								eRFID[iw1].lrWeightMeasuredCV := eWeightPackageState[1].lrWeightMeasuredCV := VIS.lrWeight1Measured;
								eRFID[iw1].lrWeightCV := eWeightPackageState[1].lrWeightCV := VIS.lrWeight1Mass:=P05_Weight.fbWeight1.lrMeasuredWeight+lrWeight1MeasurmentCorrection-lrCupWeight-lrFormWeight-lrFormWeight1RFID;	
								
								(***DIAGNOSTYKA WAGI***)
									IF eRFID[iw1].lrMinWeightCV = 0 THEN eRFID[iw1].lrMinWeightCV := ABS(eRFID[iw1].lrWeightCV); END_IF
									IF eRFID[iw1].lrMinWeightCV > ABS(eRFID[iw1].lrWeightCV)  THEN
											eRFID[iw1].lrMinWeightCV:= ABS(eRFID[iw1].lrWeightCV);
									END_IF
									IF ABS(eRFID[iw1].lrWeightCV) > eRFID[iw1].lrMaxWeightCV THEN
											eRFID[iw1].lrMaxWeightCV:= ABS(eRFID[iw1].lrWeightCV);
									END_IF
									eRFID[iw1].lrWeightDif := eRFID[iw1].lrMaxWeightCV - eRFID[iw1].lrMinWeightCV;
								(***KONIEC DIAGNOSTYKI WAGI**)
								
							
								eRFID[iw1].lrWeightSV := eWeightPackageState[1].lrWeightSV := lrWeightMassSV;
								eRFID[iw1].bWeighed := eWeightPackageState[1].bWeighed := TRUE;
								//Sprawdzanie czy doza spełnia kryteria dopuszczalenej konfekcji
								
								(*Generowaie danych do wykresów*)
								IF eRFID[iw1].nDispencerNr = 1 THEN
									VIS.lrDispencer1WeightMeasured := eRFID[iw1].lrWeightCV;	//Do wykresów HMI
									VIS.lrDispencer1DoseVolumeCV :=	eRFID[iw1].lrDoseVolumeCV;	//Do wykresów HMI
									VIS.bDispencer1WeightMeasured := TRUE; //Do wyświetlenia na ekranie głównym
								ELSE									  
									VIS.lrDispencer1WeightMeasured := VIS.lrDispencer1DoseVolumeCV := 0.0;	//Do wykresów HMI
									VIS.bDispencer1WeightMeasured := FALSE; //Do wyświetlenia na ekranie głównym
								END_IF
							
								(*Koniec generowania danych do wykresów*)
								IF 	((LREAL_TO_DINT(eRFID[iw1].lrWeightCV)-LREAL_TO_DINT(eRFID[iw1].lrWeightSV))<=(lrWeightUpperTolerance)) AND 
									((LREAL_TO_DINT(eRFID[iw1].lrWeightSV)-LREAL_TO_DINT(eRFID[iw1].lrWeightCV))<=lrWeightLowerTolerance) 
									THEN
									eRFID[iw1].bWeightOK := eWeightPackageState[1].bWeightOK := TRUE;
								END_IF	
								(*Dodatkowa informacja o wadze*)
								IF 	((LREAL_TO_DINT(eRFID[iw1].lrWeightCV)-LREAL_TO_DINT(eRFID[iw1].lrWeightSV))>lrWeightUpperTolerance) THEN
									eRFID[iw1].bWeightTooHigh := eWeightPackageState[1].bWeightTooHigh := TRUE;
								END_IF
								IF ((LREAL_TO_DINT(eRFID[iw1].lrWeightSV)-LREAL_TO_DINT(eRFID[iw1].lrWeightCV))>lrWeightLowerTolerance) THEN
									eRFID[iw1].bWeightTooLow:= eWeightPackageState[1].bWeightTooLow := TRUE;
								END_IF				
								VIS.bWeight1DoWeighting:=FALSE;
								
							END_IF																		
						ELSIF NOT bWeight1Enable THEN
							eRFID[iw1].bWeightOK 			:= eWeightPackageState[1].bWeightOK 			:=	TRUE;
							eRFID[iw1].bWeightTooHigh 		:= eWeightPackageState[1].bWeightTooHigh 		:=	FALSE;
							eRFID[iw1].bWeightTooLow		:= eWeightPackageState[1].bWeightTooLow 		:=	FALSE;
							eRFID[iw1].lrWeightMeasuredCV 	:= eWeightPackageState[1].lrWeightMeasuredCV 	:=	0;
							eRFID[iw1].lrWeightCV 			:= eWeightPackageState[1].lrWeightCV 			:=	VIS.lrWeight1Mass:=lrWeightMassSV;	
							eRFID[iw1].lrWeightSV 			:= eWeightPackageState[1].lrWeightSV 			:=	lrWeightMassSV;
							eRFID[iw1].bWeighed 			:= eWeightPackageState[1].bWeighed  			:=	FALSE;
						END_IF
						//KONIEC WARUNKI STACJI								
				ELSIF tonWeightPackageState1BnCardNumber0.Q THEN	// Jeżeli nie wykryje RFID
					VIS.bWeight1DoWeighting 			:= FALSE;
					eWeightPackageState[1].bFormPresent	:= TRUE;					
					eWeightPackageState[1].bWeightOK	:= FALSE;
					eWeightPackageState[1].bWeighed		:= TRUE;
				ELSIF tonWeightPackageState1BnNoCardNumber.Q THEN 	// Jeżeli nie ma RFID w tablicy
					itonWeightPackageState1BnNoCardNumber	:= itonWeightPackageState1BnNoCardNumber	+	1;
					VIS.bWeight1DoWeighting 			:= FALSE;
					eWeightPackageState[1].bWeightOK 	:= FALSE;
					eWeightPackageState[1].bWeighed 	:= TRUE;
				ELSE
					;
				END_IF
				
			END_FOR	
		END_IF

// Waga 2
tonWeightPackageState2BnCardNumber0			(IN:=eWeightPackageState[2].nCardNumber = 0 AND VIS.bWeight2DoWeighting OR NOT bWeight1Enable, PT:=T#5S);
tonWeightPackageState2BnNoCardNumber		(IN:=eWeightPackageState[2].nCardNumber > 0 AND VIS.bWeight2DoWeighting OR NOT bWeight1Enable, PT:=T#10S);
IF VIS.bWeight2DoWeighting THEN
			FOR iw2 := 1 TO 100 DO
				 IF eWeightPackageState[2].nCardNumber = eRFID[iw2].nCardNumber AND eWeightPackageState[2].nCardNumber > 0 THEN	
						nw2:=iw2; (*Do testów*) eRFID[nw2].bFormPresent; eRFID[nw2].bWeighed; eRFID[nw2].lrWeightMeasuredCV;
				 		//WARUNKI STACJI
						IF bWeight1Enable AND  NOT eRFID[iw2].bWeighed AND eRFID[iw2].lrWeightMeasuredCV=0 
						THEN
							//VIS.bWeight2Run:=TRUE;
							IF P05_Weight.fbWeight2.bCycleDone THEN	
								//(*Włączona waga z przeważania*) // Czyli w recepturach waga formatki wybrana na 0
								IF lrFormWeight = 0 THEN
											FOR jw2 := 1 TO 100 DO
												IF eWeightPackageState[2].nCardNumber = VIS.AnRFIDCardNumberShow[jw2] THEN	
													lrFormWeight2RFID := VIS.AnRFIDWeightShow[jw2];
													bFormWeight2Found := TRUE;
												END_IF
											END_FOR
											IF NOT bFormWeight2Found THEN
												lrFormWeight2RFID := 0;
											END_IF
											bFormWeight2Found := FALSE;
								ELSE
									lrFormWeight2RFID := 0;
								END_IF
								(**KONIEC POBIERANIE WARTOŚCI Z PRZEWAŻANIA*)
						
								eRFID[iw2].lrWeightMeasuredCV := eWeightPackageState[2].lrWeightMeasuredCV := VIS.lrWeight2Measured;
								eRFID[iw2].lrWeightCV := eWeightPackageState[2].lrWeightCV := VIS.lrWeight2Mass:=P05_Weight.fbWeight2.lrMeasuredWeight+lrWeight1MeasurmentCorrection-lrCupWeight-lrFormWeight-lrFormWeight2RFID;	
								
								(***DIAGNOSTYKA WAGI***)
									IF eRFID[iw2].lrMinWeightCV = 0 THEN eRFID[iw2].lrMinWeightCV := ABS(eRFID[iw2].lrWeightCV); END_IF
									IF eRFID[iw2].lrMinWeightCV > ABS(eRFID[iw2].lrWeightCV)  THEN
											eRFID[iw2].lrMinWeightCV:= ABS(eRFID[iw2].lrWeightCV);
									END_IF
									IF ABS(eRFID[iw2].lrWeightCV) > eRFID[iw2].lrMaxWeightCV THEN
											eRFID[iw2].lrMaxWeightCV:= ABS(eRFID[iw2].lrWeightCV);
									END_IF
									eRFID[iw2].lrWeightDif := eRFID[iw2].lrMaxWeightCV - eRFID[iw2].lrMinWeightCV;
								(***KONIEC DIAGNOSTYKI WAGI**)
								
							
								eRFID[iw2].lrWeightSV := eWeightPackageState[2].lrWeightSV := lrWeightMassSV;
								eRFID[iw2].bWeighed := eWeightPackageState[2].bWeighed:= TRUE;
								//Sprawdzanie czy doza spełnia kryteria dopuszczalenej konfekcji
								
								(*Generowaie danych do wykresów*)
								(*IF eRFID[iw2].nDispencerNr = 1 THEN
									VIS.lrDispencer1WeightMeasured := eRFID[iw2].lrWeightCV;	//Do wykresów HMI
									VIS.lrDispencer1DoseVolumeCV :=	eRFID[iw2].lrDoseVolumeCV;	//Do wykresów HMI
									VIS.bDispencer1WeightMeasured := TRUE; //Do wyświetlenia na ekranie głównym
								ELSE									  
									VIS.lrDispencer1WeightMeasured := VIS.lrDispencer1DoseVolumeCV := 0.0;	//Do wykresów HMI
									VIS.bDispencer1WeightMeasured := FALSE; //Do wyświetlenia na ekranie głównym
								END_IF*)
								IF eRFID[iw2].nDispencerNr = 2 THEN
									VIS.lrDispencer2WeightMeasured := eRFID[iw2].lrWeightCV;	//Do wykresów HMI
									VIS.lrDispencer2DoseVolumeCV :=	eRFID[iw2].lrDoseVolumeCV;	//Do wykresów HMI
									VIS.bDispencer2WeightMeasured := TRUE; //Do wyświetlenia na ekranie głównym
									IF bDosingTwoPhases THEN
										VIS.lrDispencer2DoseVolumeCV :=	eRFID[iw2].lrDoseVolumeCVSecondPhase; //Do wykresów HMI
									END_IF
								ELSE									
									VIS.lrDispencer2WeightMeasured := VIS.lrDispencer2DoseVolumeCV := 0.0;	//Do wykresów HMI
									VIS.bDispencer2WeightMeasured := FALSE; //Do wyświetlenia na ekranie głównym
								END_IF
								(*IF eRFID[iw2].nDispencerNr = 3 THEN
									VIS.lrDispencer3WeightMeasured := eRFID[iw2].lrWeightCV;	//Do wykresów HMI
									VIS.lrDispencer3DoseVolumeCV :=	eRFID[iw2].lrDoseVolumeCV;	//Do wykresów HMI
									VIS.bDispencer3WeightMeasured := TRUE; //Do wyświetlenia na ekranie głównym
								ELSE									  
									VIS.lrDispencer3WeightMeasured := VIS.lrDispencer3DoseVolumeCV := 0.0;	//Do wykresów HMI
									VIS.bDispencer3WeightMeasured := FALSE; //Do wyświetlenia na ekranie głównym
								END_IF
								
								IF eRFID[iw2].nDispencerNr = 4 THEN
									VIS.lrDispencer4WeightMeasured := eRFID[iw2].lrWeightCV;	//Do wykresów HMI
									VIS.lrDispencer4DoseVolumeCV :=	eRFID[iw2].lrDoseVolumeCV;	//Do wykresów HMI
									VIS.bDispencer4WeightMeasured := TRUE; //Do wyświetlenia na ekranie głównym
								ELSE									  
									VIS.lrDispencer4WeightMeasured := VIS.lrDispencer4DoseVolumeCV := 0.0;	//Do wykresów HMI
									VIS.bDispencer4WeightMeasured := FALSE; //Do wyświetlenia na ekranie głównym
								END_IF*)
								(*Koniec generowania danych do wykresów*)
								IF 	((LREAL_TO_DINT(eRFID[iw2].lrWeightCV)-LREAL_TO_DINT(eRFID[iw2].lrWeightSV))<=(lrWeightUpperTolerance)) AND 
									((LREAL_TO_DINT(eRFID[iw2].lrWeightSV)-LREAL_TO_DINT(eRFID[iw2].lrWeightCV))<=lrWeightLowerTolerance) 
									THEN
									eRFID[iw2].bWeightOK := eWeightPackageState[2].bWeightOK := TRUE;
								END_IF	
								(*Dodatkowa informacja o wadze*)
								IF 	((LREAL_TO_DINT(eRFID[iw2].lrWeightCV)-LREAL_TO_DINT(eRFID[iw2].lrWeightSV))>lrWeightUpperTolerance) THEN
									eRFID[iw2].bWeightTooHigh := eWeightPackageState[2].bWeightTooHigh := TRUE;
								END_IF
								IF ((LREAL_TO_DINT(eRFID[iw2].lrWeightSV)-LREAL_TO_DINT(eRFID[iw2].lrWeightCV))>lrWeightLowerTolerance) THEN
									eRFID[iw2].bWeightTooLow:= eWeightPackageState[2].bWeightTooLow := TRUE;
								END_IF	
								
								VIS.bWeight2DoWeighting:=FALSE;
								
							END_IF																		
						ELSIF NOT bWeight1Enable THEN
							eRFID[iw2].bWeightOK := eWeightPackageState[2].bWeightOK := TRUE;
							eRFID[iw2].bWeightTooHigh := eWeightPackageState[2].bWeightTooHigh := FALSE;
							eRFID[iw2].bWeightTooLow:= eWeightPackageState[2].bWeightTooLow := FALSE;
							eRFID[iw2].lrWeightMeasuredCV := eWeightPackageState[2].lrWeightMeasuredCV := 0;
							eRFID[iw2].lrWeightCV := eWeightPackageState[2].lrWeightCV :=VIS.lrWeight2Mass:=lrWeightMassSV;	
							eRFID[iw2].lrWeightSV := eWeightPackageState[2].lrWeightSV :=lrWeightMassSV;
							eRFID[iw2].bWeighed := eWeightPackageState[2].bWeighed  := FALSE;
						END_IF
						//KONIEC WARUNKI STACJI								
				ELSIF tonWeightPackageState2BnCardNumber0.Q THEN	// Jeżeli nie wykryje RFID
					VIS.bWeight2DoWeighting 					:= FALSE;
					eWeightPackageState[2].bFormPresent	:= TRUE;	//Dp		
					eWeightPackageState[2].bWeightOK	:= FALSE;
					eWeightPackageState[2].bWeighed		:= TRUE;
				ELSIF tonWeightPackageState2BnNoCardNumber.Q THEN 	// Jeżeli nie ma RFID w tablicy
					itonWeightPackageState2BnNoCardNumber	:= itonWeightPackageState2BnNoCardNumber	+	1;					
					VIS.bWeight2DoWeighting 					:= FALSE;
					eWeightPackageState[2].bWeightOK 	:= FALSE;
					eWeightPackageState[2].bWeighed 	:= TRUE;
				ELSE
					;
				END_IF
				
			END_FOR	
		END_IF

// Waga 3
tonWeightPackageState3BnCardNumber0			(IN:=eWeightPackageState[3].nCardNumber = 0 AND VIS.bWeight3DoWeighting OR NOT bWeight1Enable, PT:=T#5S);
tonWeightPackageState3BnNoCardNumber		(IN:=eWeightPackageState[3].nCardNumber > 0 AND VIS.bWeight3DoWeighting OR NOT bWeight1Enable, PT:=T#10S);
IF VIS.bWeight3DoWeighting THEN
			FOR iw3 := 1 TO 100 DO
				 IF eWeightPackageState[3].nCardNumber = eRFID[iw3].nCardNumber AND eWeightPackageState[3].nCardNumber > 0 THEN	
						nw3:=iw3; (*Do testów*) eRFID[nw3].bFormPresent; eRFID[nw3].bWeighed; eRFID[nw3].lrWeightMeasuredCV;
				 		//WARUNKI STACJI
						IF bWeight1Enable AND NOT eRFID[iw3].bWeighed AND eRFID[iw3].lrWeightMeasuredCV=0 
						THEN
						//	VIS.bWeight3Run:=TRUE;
							IF P05_Weight.fbWeight3.bCycleDone THEN	
								//(*Włączona waga z przeważania*) // Czyli w recepturach waga formatki wybrana na 0
								IF lrFormWeight = 0 THEN
											FOR jw3 := 1 TO 100 DO
												IF eWeightPackageState[3].nCardNumber = VIS.AnRFIDCardNumberShow[jw3] THEN	
													lrFormWeight3RFID := VIS.AnRFIDWeightShow[jw3];
													bFormWeight3Found := TRUE;
												END_IF
											END_FOR
											IF NOT bFormWeight3Found THEN
												lrFormWeight3RFID := 0;
											END_IF
											bFormWeight3Found := FALSE;
								ELSE
									lrFormWeight3RFID := 0;
								END_IF
								(**KONIEC POBIERANIE WARTOŚCI Z PRZEWAŻANIA*)
						
								eRFID[iw3].lrWeightMeasuredCV := eWeightPackageState[3].lrWeightMeasuredCV := VIS.lrWeight3Measured;
								eRFID[iw3].lrWeightCV := eWeightPackageState[3].lrWeightCV := VIS.lrWeight3Mass:=P05_Weight.fbWeight3.lrMeasuredWeight+lrWeight1MeasurmentCorrection-lrCupWeight-lrFormWeight-lrFormWeight3RFID;	
								
								(***DIAGNOSTYKA WAGI***)
									IF eRFID[iw3].lrMinWeightCV = 0 THEN eRFID[iw3].lrMinWeightCV := ABS(eRFID[iw3].lrWeightCV); END_IF
									IF eRFID[iw3].lrMinWeightCV > ABS(eRFID[iw3].lrWeightCV)  THEN
											eRFID[iw3].lrMinWeightCV:= ABS(eRFID[iw3].lrWeightCV);
									END_IF
									IF ABS(eRFID[iw3].lrWeightCV) > eRFID[iw3].lrMaxWeightCV THEN
											eRFID[iw3].lrMaxWeightCV:= ABS(eRFID[iw3].lrWeightCV);
									END_IF
									eRFID[iw3].lrWeightDif := eRFID[iw3].lrMaxWeightCV - eRFID[iw3].lrMinWeightCV;
								(***KONIEC DIAGNOSTYKI WAGI**)
								
							
								eRFID[iw3].lrWeightSV := eWeightPackageState[3].lrWeightSV := lrWeightMassSV;
								eRFID[iw3].bWeighed := eWeightPackageState[3].bWeighed := TRUE;
								//Sprawdzanie czy doza spełnia kryteria dopuszczalenej konfekcji
								
								(*Generowaie danych do wykresów*)
								(*IF eRFID[iw3].nDispencerNr = 1 THEN
									VIS.lrDispencer1WeightMeasured := eRFID[iw3].lrWeightCV;	//Do wykresów HMI
									VIS.lrDispencer1DoseVolumeCV :=	eRFID[iw3].lrDoseVolumeCV;	//Do wykresów HMI
									VIS.bDispencer1WeightMeasured := TRUE; //Do wyświetlenia na ekranie głównym
								ELSE									  
									VIS.lrDispencer1WeightMeasured := VIS.lrDispencer1DoseVolumeCV := 0.0;	//Do wykresów HMI
									VIS.bDispencer1WeightMeasured := FALSE; //Do wyświetlenia na ekranie głównym
								END_IF
								IF eRFID[iw3].nDispencerNr = 2 THEN
									VIS.lrDispencer2WeightMeasured := eRFID[iw3].lrWeightCV;	//Do wykresów HMI
									VIS.lrDispencer2DoseVolumeCV :=	eRFID[iw3].lrDoseVolumeCV;	//Do wykresów HMI
									VIS.bDispencer2WeightMeasured := TRUE; //Do wyświetlenia na ekranie głównym
									IF bDosingTwoPhases THEN
										VIS.lrDispencer2DoseVolumeCV :=	eRFID[iw3].lrDoseVolumeCVSecondPhase; //Do wykresów HMI
									END_IF
								ELSE									
									VIS.lrDispencer2WeightMeasured := VIS.lrDispencer2DoseVolumeCV := 0.0;	//Do wykresów HMI
									VIS.bDispencer2WeightMeasured := FALSE; //Do wyświetlenia na ekranie głównym
								END_IF*)
								IF eRFID[iw3].nDispencerNr = 3 THEN
									VIS.lrDispencer3WeightMeasured := eRFID[iw3].lrWeightCV;	//Do wykresów HMI
									VIS.lrDispencer3DoseVolumeCV :=	eRFID[iw3].lrDoseVolumeCV;	//Do wykresów HMI
									VIS.bDispencer3WeightMeasured := TRUE; //Do wyświetlenia na ekranie głównym
								ELSE									  
									VIS.lrDispencer3WeightMeasured := VIS.lrDispencer3DoseVolumeCV := 0.0;	//Do wykresów HMI
									VIS.bDispencer3WeightMeasured := FALSE; //Do wyświetlenia na ekranie głównym
								END_IF
								
								(*IF eRFID[iw3].nDispencerNr = 4 THEN
									VIS.lrDispencer4WeightMeasured := eRFID[iw3].lrWeightCV;	//Do wykresów HMI
									VIS.lrDispencer4DoseVolumeCV :=	eRFID[iw3].lrDoseVolumeCV;	//Do wykresów HMI
									VIS.bDispencer4WeightMeasured := TRUE; //Do wyświetlenia na ekranie głównym
								ELSE									  
									VIS.lrDispencer4WeightMeasured := VIS.lrDispencer4DoseVolumeCV := 0.0;	//Do wykresów HMI
									VIS.bDispencer4WeightMeasured := FALSE; //Do wyświetlenia na ekranie głównym
								END_IF	*)						
								(*Koniec generowania danych do wykresów*)
								IF 	((LREAL_TO_DINT(eRFID[iw3].lrWeightCV)-LREAL_TO_DINT(eRFID[iw3].lrWeightSV))<=(lrWeightUpperTolerance)) AND 
									((LREAL_TO_DINT(eRFID[iw3].lrWeightSV)-LREAL_TO_DINT(eRFID[iw3].lrWeightCV))<=lrWeightLowerTolerance) 
									THEN
									eRFID[iw3].bWeightOK := eWeightPackageState[3].bWeightOK := TRUE;
								END_IF	
								(*Dodatkowa informacja o wadze*)
								
								IF 	((LREAL_TO_DINT(eRFID[iw3].lrWeightCV)-LREAL_TO_DINT(eRFID[iw3].lrWeightSV))>lrWeightUpperTolerance) THEN
									eRFID[iw3].bWeightTooHigh := eWeightPackageState[3].bWeightTooHigh := TRUE;
								END_IF
								IF ((LREAL_TO_DINT(eRFID[iw3].lrWeightSV)-LREAL_TO_DINT(eRFID[iw3].lrWeightCV))>lrWeightLowerTolerance) THEN
									eRFID[iw3].bWeightTooLow:= eWeightPackageState[3].bWeightTooLow := TRUE;
								END_IF	
								
								VIS.bWeight3DoWeighting:=FALSE;
								
							END_IF																		
						ELSIF NOT bWeight1Enable THEN
							eRFID[iw3].bWeightOK := eWeightPackageState[3].bWeightOK := TRUE;
							eRFID[iw3].bWeightTooHigh := eWeightPackageState[3].bWeightTooHigh := FALSE;
							eRFID[iw3].bWeightTooLow:= eWeightPackageState[3].bWeightTooLow := FALSE;
							eRFID[iw3].lrWeightMeasuredCV := eWeightPackageState[3].lrWeightMeasuredCV := 0;
							eRFID[iw3].lrWeightCV := eWeightPackageState[3].lrWeightCV :=VIS.lrWeight3Mass:=lrWeightMassSV;	
							eRFID[iw3].lrWeightSV := eWeightPackageState[3].lrWeightSV :=lrWeightMassSV;
							eRFID[iw3].bWeighed := eWeightPackageState[3].bWeighed  := FALSE;
						END_IF
						//KONIEC WARUNKI STACJI								
				ELSIF tonWeightPackageState3BnCardNumber0.Q THEN	// Jeżeli nie wykryje RFID
					VIS.bWeight3DoWeighting 					:= FALSE;
					eWeightPackageState[3].bFormPresent	:= TRUE;	//Dp		
					eWeightPackageState[3].bWeightOK 	:= FALSE;
					eWeightPackageState[3].bWeighed 	:= TRUE;
				ELSIF tonWeightPackageState3BnNoCardNumber.Q THEN 	// Jeżeli nie ma RFID w tablicy
					itonWeightPackageState3BnNoCardNumber	:= itonWeightPackageState3BnNoCardNumber	+	1;						
					VIS.bWeight3DoWeighting 					:= FALSE;
					eWeightPackageState[3].bWeightOK 	:= FALSE;
					eWeightPackageState[3].bWeighed 	:= TRUE;
				ELSE
					;
				END_IF
				
			END_FOR	
		END_IF

// Waga 4
tonWeightPackageState4BnCardNumber0			(IN:=eWeightPackageState[4].nCardNumber = 0 AND VIS.bWeight4DoWeighting OR NOT bWeight1Enable, PT:=T#5S);
tonWeightPackageState4BnNoCardNumber		(IN:=eWeightPackageState[4].nCardNumber > 0 AND VIS.bWeight4DoWeighting OR NOT bWeight1Enable, PT:=T#10S);
IF VIS.bWeight4DoWeighting THEN
			FOR iw4 := 1 TO 100 DO
				 IF eWeightPackageState[4].nCardNumber = eRFID[iw4].nCardNumber AND eWeightPackageState[4].nCardNumber > 0 THEN	
						nw4:=iw4; (*Do testów*) eRFID[nw4].bFormPresent; eRFID[nw4].bWeighed; eRFID[nw4].lrWeightMeasuredCV;
				 		//WARUNKI STACJI
						IF bWeight1Enable AND NOT eRFID[iw4].bWeighed AND eRFID[iw4].lrWeightMeasuredCV=0 
						THEN
							//VIS.bWeight4Run:=TRUE;
							IF P05_Weight.fbWeight4.bCycleDone THEN	
								//(*Włączona waga z przeważania*) // Czyli w recepturach waga formatki wybrana na 0
								IF lrFormWeight = 0 THEN
											FOR jw4 := 1 TO 100 DO
												IF eWeightPackageState[4].nCardNumber = VIS.AnRFIDCardNumberShow[jw4] THEN	
													lrFormWeight4RFID := VIS.AnRFIDWeightShow[jw4];
													bFormWeight4Found := TRUE;
												END_IF
											END_FOR
											IF NOT bFormWeight4Found THEN
												lrFormWeight4RFID := 0;
											END_IF
											bFormWeight4Found := FALSE;
								ELSE
									lrFormWeight4RFID := 0;
								END_IF
								(**KONIEC POBIERANIE WARTOŚCI Z PRZEWAŻANIA*)
						
								eRFID[iw4].lrWeightMeasuredCV := eWeightPackageState[4].lrWeightMeasuredCV := VIS.lrWeight4Measured;
								eRFID[iw4].lrWeightCV := eWeightPackageState[4].lrWeightCV := VIS.lrWeight4Mass:=P05_Weight.fbWeight4.lrMeasuredWeight+lrWeight1MeasurmentCorrection-lrCupWeight-lrFormWeight-lrFormWeight4RFID;	
								
								(***DIAGNOSTYKA WAGI***)
									IF eRFID[iw4].lrMinWeightCV = 0 THEN eRFID[iw4].lrMinWeightCV := ABS(eRFID[iw4].lrWeightCV); END_IF
									IF eRFID[iw4].lrMinWeightCV > ABS(eRFID[iw4].lrWeightCV)  THEN
											eRFID[iw4].lrMinWeightCV:= ABS(eRFID[iw4].lrWeightCV);
									END_IF
									IF ABS(eRFID[iw4].lrWeightCV) > eRFID[iw4].lrMaxWeightCV THEN
											eRFID[iw4].lrMaxWeightCV:= ABS(eRFID[iw4].lrWeightCV);
									END_IF
									eRFID[iw4].lrWeightDif := eRFID[iw4].lrMaxWeightCV - eRFID[iw4].lrMinWeightCV;
								(***KONIEC DIAGNOSTYKI WAGI**)
								
							
								eRFID[iw4].lrWeightSV := eWeightPackageState[4].lrWeightSV := lrWeightMassSV;
								eRFID[iw4].bWeighed := eWeightPackageState[4].bWeighed := TRUE;
								//Sprawdzanie czy doza spełnia kryteria dopuszczalenej konfekcji
								
								(*Generowaie danych do wykresów*)
								(*IF eRFID[iw4].nDispencerNr = 1 THEN
									VIS.lrDispencer1WeightMeasured := eRFID[iw4].lrWeightCV;	//Do wykresów HMI
									VIS.lrDispencer1DoseVolumeCV :=	eRFID[iw4].lrDoseVolumeCV;	//Do wykresów HMI
									VIS.bDispencer1WeightMeasured := TRUE; //Do wyświetlenia na ekranie głównym
								ELSE									  
									VIS.lrDispencer1WeightMeasured := VIS.lrDispencer1DoseVolumeCV := 0.0;	//Do wykresów HMI
									VIS.bDispencer1WeightMeasured := FALSE; //Do wyświetlenia na ekranie głównym
								END_IF
								IF eRFID[iw4].nDispencerNr = 2 THEN
									VIS.lrDispencer2WeightMeasured := eRFID[iw4].lrWeightCV;	//Do wykresów HMI
									VIS.lrDispencer2DoseVolumeCV :=	eRFID[iw4].lrDoseVolumeCV;	//Do wykresów HMI
									VIS.bDispencer2WeightMeasured := TRUE; //Do wyświetlenia na ekranie głównym
									IF bDosingTwoPhases THEN
										VIS.lrDispencer2DoseVolumeCV :=	eRFID[iw4].lrDoseVolumeCVSecondPhase; //Do wykresów HMI
									END_IF
								ELSE									
									VIS.lrDispencer2WeightMeasured := VIS.lrDispencer2DoseVolumeCV := 0.0;	//Do wykresów HMI
									VIS.bDispencer2WeightMeasured := FALSE; //Do wyświetlenia na ekranie głównym
								END_IF
								IF eRFID[iw4].nDispencerNr = 3 THEN
									VIS.lrDispencer3WeightMeasured := eRFID[iw4].lrWeightCV;	//Do wykresów HMI
									VIS.lrDispencer3DoseVolumeCV :=	eRFID[iw4].lrDoseVolumeCV;	//Do wykresów HMI
									VIS.bDispencer3WeightMeasured := TRUE; //Do wyświetlenia na ekranie głównym
								ELSE									  
									VIS.lrDispencer3WeightMeasured := VIS.lrDispencer3DoseVolumeCV := 0.0;	//Do wykresów HMI
									VIS.bDispencer3WeightMeasured := FALSE; //Do wyświetlenia na ekranie głównym
								END_IF*)
								
								IF eRFID[iw4].nDispencerNr = 4 THEN
									VIS.lrDispencer4WeightMeasured := eRFID[iw4].lrWeightCV;	//Do wykresów HMI
									VIS.lrDispencer4DoseVolumeCV :=	eRFID[iw4].lrDoseVolumeCV;	//Do wykresów HMI
									VIS.bDispencer4WeightMeasured := TRUE; //Do wyświetlenia na ekranie głównym
								ELSE									  
									VIS.lrDispencer4WeightMeasured := VIS.lrDispencer4DoseVolumeCV := 0.0;	//Do wykresów HMI
									VIS.bDispencer4WeightMeasured := FALSE; //Do wyświetlenia na ekranie głównym
								END_IF
								
								(*Koniec generowania danych do wykresów*)
								IF 	((LREAL_TO_DINT(eRFID[iw4].lrWeightCV)-LREAL_TO_DINT(eRFID[iw4].lrWeightSV))<=(lrWeightUpperTolerance)) AND 
									((LREAL_TO_DINT(eRFID[iw4].lrWeightSV)-LREAL_TO_DINT(eRFID[iw4].lrWeightCV))<=lrWeightLowerTolerance) 
									THEN
									eRFID[iw4].bWeightOK := eWeightPackageState[4].bWeightOK := TRUE;
								END_IF	
								(*Dodatkowa informacja o wadze*)
								IF 	((LREAL_TO_DINT(eRFID[iw4].lrWeightCV)-LREAL_TO_DINT(eRFID[iw4].lrWeightSV))>lrWeightUpperTolerance) THEN
									eRFID[iw4].bWeightTooHigh := eWeightPackageState[4].bWeightTooHigh := TRUE;
								END_IF
								IF ((LREAL_TO_DINT(eRFID[iw4].lrWeightSV)-LREAL_TO_DINT(eRFID[iw4].lrWeightCV))>lrWeightLowerTolerance) THEN
									eRFID[iw4].bWeightTooLow:= eWeightPackageState[4].bWeightTooLow := TRUE;
								END_IF

							VIS.bWeight4DoWeighting:=FALSE;
	
							END_IF																		
						ELSIF NOT bWeight1Enable THEN
							eRFID[iw4].bWeightOK := eWeightPackageState[4].bWeightOK := TRUE;
							eRFID[iw4].bWeightTooHigh := eWeightPackageState[4].bWeightTooHigh := FALSE;
							eRFID[iw4].bWeightTooLow:= eWeightPackageState[4].bWeightTooLow := FALSE;
							eRFID[iw4].lrWeightMeasuredCV := eWeightPackageState[4].lrWeightMeasuredCV := 0;
							eRFID[iw4].lrWeightCV := eWeightPackageState[4].lrWeightCV :=VIS.lrWeight4Mass:=lrWeightMassSV;	
							eRFID[iw4].lrWeightSV := eWeightPackageState[4].lrWeightSV :=lrWeightMassSV;
							eRFID[iw4].bWeighed := eWeightPackageState[4].bWeighed  := FALSE;
						END_IF
						//KONIEC WARUNKI STACJI								
				ELSIF tonWeightPackageState4BnCardNumber0.Q THEN	// Jeżeli nie wykryje RFID
					VIS.bWeight4DoWeighting 					:= FALSE;
					eWeightPackageState[4].bFormPresent	:= TRUE;	//Dp		
					eWeightPackageState[4].bWeightOK 	:= FALSE;
					eWeightPackageState[4].bWeighed 	:= TRUE;
				ELSIF tonWeightPackageState4BnNoCardNumber.Q THEN 	// Jeżeli nie ma RFID w tablicy
					itonWeightPackageState4BnNoCardNumber	:= itonWeightPackageState4BnNoCardNumber	+	1;							
					VIS.bWeight4DoWeighting 					:= FALSE;
					eWeightPackageState[4].bWeightOK 	:= FALSE;
					eWeightPackageState[4].bWeighed 	:= TRUE;
				ELSE
					;
				END_IF
				
			END_FOR	
		END_IF										
(********************KONIEC WAZENIA**************************)
(************************************************************)

(********************Ważenie przy dwufazie**************************)
(*******************************************************************)






// Waga 5 - 1 waga na drugiej fazie
tonWeightPackageState5BnCardNumber0			(IN:=eWeightPackage2PhasePackageState[1].nCardNumber = 0 AND VIS.bWeight5DoWeighting OR NOT bWeight1Enable, PT:=T#3S);
tonWeightPackageState5BnNoCardNumber		(IN:=eWeightPackage2PhasePackageState[1].nCardNumber > 0 AND VIS.bWeight5DoWeighting OR NOT bWeight1Enable, PT:=T#10S);
IF VIS.bWeight5DoWeighting THEN
			FOR iw5 := 1 TO 100 DO
				 IF eWeightPackage2PhasePackageState[1].nCardNumber = eRFID[iw5].nCardNumber AND eWeightPackage2PhasePackageState[1].nCardNumber > 0 THEN	
						nw5:=iw5; (*Do testów*) eRFID[nw5].bFormPresent; eRFID[nw5].bWeighed; eRFID[nw5].lrWeightMeasuredCV;
				 		//WARUNKI STACJI
						IF bWeight1Enable AND NOT eRFID[iw5].bWeighed AND eRFID[iw5].lrWeightMeasuredCV=0 
						THEN
							//VIS.bWeight4Run:=TRUE;
							IF P05_Weight.fbWeight5.bCycleDone THEN	
								//(*Włączona waga z przeważania*) // Czyli w recepturach waga formatki wybrana na 0
								IF lrFormWeight = 0 THEN
											FOR jw5 := 1 TO 100 DO
												IF eWeightPackage2PhasePackageState[1].nCardNumber = VIS.AnRFIDCardNumberShow[jw5] THEN	
													lrFormWeight5RFID := VIS.AnRFIDWeightShow[jw5];
													bFormWeight5Found := TRUE;
												END_IF
											END_FOR
											IF NOT bFormWeight5Found THEN
												lrFormWeight5RFID := 0;
											END_IF
											bFormWeight5Found := FALSE;
								ELSE
									lrFormWeight5RFID := 0;
								END_IF
								(**KONIEC POBIERANIE WARTOŚCI Z PRZEWAŻANIA*)
						
								eRFID[iw5].lrWeightMeasuredCV := eWeightPackage2PhasePackageState[1].lrWeightMeasuredCV := VIS.lrWeight5Measured;
								eRFID[iw5].lrWeightCV := eWeightPackage2PhasePackageState[1].lrWeightCV := VIS.lrWeight5Mass:=P05_Weight.fbWeight5.lrMeasuredWeight+lrWeight1MeasurmentCorrection-lrCupWeight-lrFormWeight-lrFormWeight5RFID;	
								
								(***DIAGNOSTYKA WAGI***)
									IF eRFID[iw5].lrMinWeightCV = 0 THEN eRFID[iw5].lrMinWeightCV := ABS(eRFID[iw5].lrWeightCV); END_IF
									IF eRFID[iw5].lrMinWeightCV > ABS(eRFID[iw5].lrWeightCV)  THEN
											eRFID[iw5].lrMinWeightCV:= ABS(eRFID[iw5].lrWeightCV);
									END_IF
									IF ABS(eRFID[iw5].lrWeightCV) > eRFID[iw5].lrMaxWeightCV THEN
											eRFID[iw5].lrMaxWeightCV:= ABS(eRFID[iw5].lrWeightCV);
									END_IF
									eRFID[iw5].lrWeightDif := eRFID[iw5].lrMaxWeightCV - eRFID[iw5].lrMinWeightCV;
								(***KONIEC DIAGNOSTYKI WAGI**)
								
							
								eRFID[iw5].lrWeightSV := eWeightPackage2PhasePackageState[1].lrWeightSV := lrWeightMassSV;
								eRFID[iw5].bWeighed := eWeightPackage2PhasePackageState[1].bWeighed := TRUE;
								//Sprawdzanie czy doza spełnia kryteria dopuszczalenej konfekcji
								
								(*Generowaie danych do wykresów*)
								VIS.lrDispencer1WeightMeasured 	:= eRFID[iw5].lrWeightCV;	//Do wykresów HMI
								//VIS.lrDispencer1DoseVolumeCV 	:=	eRFID[iw5].lrDoseVolumeCV;	//Do wykresów HMI
								
								IF eRFID[iw5].nDispencerNr = 1 THEN
									VIS.lrDispencer1DoseVolumeCV :=	eRFID[iw5].lrDoseVolumeCV;	
								ELSIF eRFID[iw5].nDispencerNr = 2 THEN
									VIS.lrDispencer2DoseVolumeCV :=	eRFID[iw5].lrDoseVolumeCV;
								ELSIF eRFID[iw5].nDispencerNr = 3 THEN
									VIS.lrDispencer3DoseVolumeCV :=	eRFID[iw5].lrDoseVolumeCVSecondPhase;
								ELSIF eRFID[iw5].nDispencerNr = 4 THEN
									VIS.lrDispencer4DoseVolumeCV :=	eRFID[iw5].lrDoseVolumeCVSecondPhase;	
								ELSE									  
									VIS.lrDispencer4DoseVolumeCV := 0.0;
								END_IF	
			
								(*IF eRFID[iw5].nDispencerNr = 1 THEN
									VIS.lrDispencer1WeightMeasured := eRFID[iw5].lrWeightCV;	//Do wykresów HMI
									VIS.lrDispencer1DoseVolumeCV :=	eRFID[iw5].lrDoseVolumeCV;	//Do wykresów HMI
									VIS.bDispencer1WeightMeasured := TRUE; //Do wyświetlenia na ekranie głównym
								ELSE									  
									VIS.lrDispencer1WeightMeasured := VIS.lrDispencer1DoseVolumeCV := 0.0;	//Do wykresów HMI
									VIS.bDispencer1WeightMeasured := FALSE; //Do wyświetlenia na ekranie głównym
								END_IF
								IF eRFID[iw5].nDispencerNr = 2 THEN
									VIS.lrDispencer2WeightMeasured := eRFID[iw5].lrWeightCV;	//Do wykresów HMI
									VIS.lrDispencer2DoseVolumeCV :=	eRFID[iw5].lrDoseVolumeCV;	//Do wykresów HMI
									VIS.bDispencer2WeightMeasured := TRUE; //Do wyświetlenia na ekranie głównym
									IF bDosingTwoPhases THEN
										VIS.lrDispencer2DoseVolumeCV :=	eRFID[iw5].lrDoseVolumeCVSecondPhase; //Do wykresów HMI
									END_IF
								ELSE									
									VIS.lrDispencer2WeightMeasured := VIS.lrDispencer2DoseVolumeCV := 0.0;	//Do wykresów HMI
									VIS.bDispencer2WeightMeasured := FALSE; //Do wyświetlenia na ekranie głównym
								END_IF
								IF eRFID[iw5].nDispencerNr = 3 THEN
									VIS.lrDispencer3WeightMeasured := eRFID[iw5].lrWeightCV;	//Do wykresów HMI
									VIS.lrDispencer3DoseVolumeCV :=	eRFID[iw5].lrDoseVolumeCV;	//Do wykresów HMI
									VIS.bDispencer3WeightMeasured := TRUE; //Do wyświetlenia na ekranie głównym
								ELSE									  
									VIS.lrDispencer3WeightMeasured := VIS.lrDispencer3DoseVolumeCV := 0.0;	//Do wykresów HMI
									VIS.bDispencer3WeightMeasured := FALSE; //Do wyświetlenia na ekranie głównym
								END_IF
								
								IF eRFID[iw5].nDispencerNr = 4 THEN
									VIS.lrDispencer4WeightMeasured := eRFID[iw5].lrWeightCV;	//Do wykresów HMI
									VIS.lrDispencer4DoseVolumeCV :=	eRFID[iw5].lrDoseVolumeCV;	//Do wykresów HMI
									VIS.bDispencer4WeightMeasured := TRUE; //Do wyświetlenia na ekranie głównym
								ELSE									  
									VIS.lrDispencer4WeightMeasured := VIS.lrDispencer4DoseVolumeCV := 0.0;	//Do wykresów HMI
									VIS.bDispencer4WeightMeasured := FALSE; //Do wyświetlenia na ekranie głównym
								END_IF*)
								
								
								
								(*Koniec generowania danych do wykresów*)
								IF 	((LREAL_TO_DINT(eRFID[iw5].lrWeightCV)-LREAL_TO_DINT(eRFID[iw5].lrWeightSV))<=(lrWeightUpperTolerance)) AND 
									((LREAL_TO_DINT(eRFID[iw5].lrWeightSV)-LREAL_TO_DINT(eRFID[iw5].lrWeightCV))<=lrWeightLowerTolerance) 
									THEN
									eRFID[iw5].bWeightOK := eWeightPackage2PhasePackageState[1].bWeightOK := TRUE;
								END_IF	
								(*Dodatkowa informacja o wadze*)
								IF 	((LREAL_TO_DINT(eRFID[iw5].lrWeightCV)-LREAL_TO_DINT(eRFID[iw5].lrWeightSV))>lrWeightUpperTolerance) THEN
									eRFID[iw5].bWeightTooHigh := eWeightPackage2PhasePackageState[1].bWeightTooHigh := TRUE;
								END_IF
								IF ((LREAL_TO_DINT(eRFID[iw5].lrWeightSV)-LREAL_TO_DINT(eRFID[iw5].lrWeightCV))>lrWeightLowerTolerance) THEN
									eRFID[iw5].bWeightTooLow:= eWeightPackage2PhasePackageState[1].bWeightTooLow := TRUE;
								END_IF

							VIS.bWeight5DoWeighting:=FALSE;
	
							END_IF																		
						ELSIF NOT bWeight1Enable THEN
							eRFID[iw5].bWeightOK := eWeightPackage2PhasePackageState[1].bWeightOK := TRUE;
							eRFID[iw5].bWeightTooHigh := eWeightPackage2PhasePackageState[1].bWeightTooHigh := FALSE;
							eRFID[iw5].bWeightTooLow:= eWeightPackage2PhasePackageState[1].bWeightTooLow := FALSE;
							eRFID[iw5].lrWeightMeasuredCV := eWeightPackage2PhasePackageState[1].lrWeightMeasuredCV := 0;
							eRFID[iw5].lrWeightCV := eWeightPackage2PhasePackageState[1].lrWeightCV :=VIS.lrWeight5Mass:=lrWeightMassSV;	
							eRFID[iw5].lrWeightSV := eWeightPackage2PhasePackageState[1].lrWeightSV :=lrWeightMassSV;
							eRFID[iw5].bWeighed := eWeightPackage2PhasePackageState[1].bWeighed  := FALSE;
						END_IF
						//KONIEC WARUNKI STACJI								
				ELSIF tonWeightPackageState5BnCardNumber0.Q THEN	// Jeżeli nie wykryje RFID
					VIS.bWeight5DoWeighting 					:= FALSE;
					eWeightPackage2PhasePackageState[1].bFormPresent	:= TRUE;	//Dp		
					eWeightPackage2PhasePackageState[1].bWeightOK 	:= FALSE;
					eWeightPackage2PhasePackageState[1].bWeighed 	:= TRUE;
				ELSIF tonWeightPackageState5BnNoCardNumber.Q THEN 	// Jeżeli nie ma RFID w tablicy
					VIS.bWeight5DoWeighting 					:= FALSE;
					eWeightPackage2PhasePackageState[1].bWeightOK 	:= FALSE;
					eWeightPackage2PhasePackageState[1].bWeighed 	:= TRUE;
				ELSE
					;
				END_IF
				
			END_FOR	
		END_IF	

// Waga 6 - 2 waga na drugiej fazie
tonWeightPackageState6BnCardNumber0			(IN:=eWeightPackage2PhasePackageState[2].nCardNumber = 0 AND VIS.bWeight6DoWeighting OR NOT bWeight1Enable, PT:=T#3S);
tonWeightPackageState6BnNoCardNumber		(IN:=eWeightPackage2PhasePackageState[2].nCardNumber > 0 AND VIS.bWeight6DoWeighting OR NOT bWeight1Enable, PT:=T#10S);
IF VIS.bWeight6DoWeighting THEN
			FOR iw6 := 1 TO 100 DO
				 IF eWeightPackage2PhasePackageState[2].nCardNumber = eRFID[iw6].nCardNumber AND eWeightPackage2PhasePackageState[2].nCardNumber > 0 THEN	
						nw6:=iw6; (*Do testów*) eRFID[nw6].bFormPresent; eRFID[nw6].bWeighed; eRFID[nw6].lrWeightMeasuredCV;
				 		//WARUNKI STACJI
						IF bWeight1Enable AND NOT eRFID[iw6].bWeighed AND eRFID[iw6].lrWeightMeasuredCV=0 
						THEN
							//VIS.bWeight4Run:=TRUE;
							IF P05_Weight.fbWeight6.bCycleDone THEN	
								//(*Włączona waga z przeważania*) // Czyli w recepturach waga formatki wybrana na 0
								IF lrFormWeight = 0 THEN
											FOR jw6 := 1 TO 100 DO
												IF eWeightPackage2PhasePackageState[2].nCardNumber = VIS.AnRFIDCardNumberShow[jw6] THEN	
													lrFormWeight6RFID := VIS.AnRFIDWeightShow[jw6];
													bFormWeight6Found := TRUE;
												END_IF
											END_FOR
											IF NOT bFormWeight6Found THEN
												lrFormWeight6RFID := 0;
											END_IF
											bFormWeight6Found := FALSE;
								ELSE
									lrFormWeight6RFID := 0;
								END_IF
								(**KONIEC POBIERANIE WARTOŚCI Z PRZEWAŻANIA*)
						
								eRFID[iw6].lrWeightMeasuredCV := eWeightPackage2PhasePackageState[2].lrWeightMeasuredCV := VIS.lrWeight6Measured;
								eRFID[iw6].lrWeightCV := eWeightPackage2PhasePackageState[2].lrWeightCV := VIS.lrWeight6Mass:=P05_Weight.fbWeight6.lrMeasuredWeight+lrWeight1MeasurmentCorrection-lrCupWeight-lrFormWeight-lrFormWeight6RFID;	
								
								(***DIAGNOSTYKA WAGI***)
									IF eRFID[iw6].lrMinWeightCV = 0 THEN eRFID[iw6].lrMinWeightCV := ABS(eRFID[iw6].lrWeightCV); END_IF
									IF eRFID[iw6].lrMinWeightCV > ABS(eRFID[iw6].lrWeightCV)  THEN
											eRFID[iw6].lrMinWeightCV:= ABS(eRFID[iw6].lrWeightCV);
									END_IF
									IF ABS(eRFID[iw6].lrWeightCV) > eRFID[iw6].lrMaxWeightCV THEN
											eRFID[iw6].lrMaxWeightCV:= ABS(eRFID[iw6].lrWeightCV);
									END_IF
									eRFID[iw6].lrWeightDif := eRFID[iw6].lrMaxWeightCV - eRFID[iw6].lrMinWeightCV;
								(***KONIEC DIAGNOSTYKI WAGI**)
								
							
								eRFID[iw6].lrWeightSV := eWeightPackage2PhasePackageState[2].lrWeightSV := lrWeightMassSV;
								eRFID[iw6].bWeighed := eWeightPackage2PhasePackageState[2].bWeighed := TRUE;
								//Sprawdzanie czy doza spełnia kryteria dopuszczalenej konfekcji
								
								(*Generowaie danych do wykresów*)
								
								VIS.lrDispencer2WeightMeasured 	:= eRFID[iw6].lrWeightCV;	//Do wykresów HMI
								//VIS.lrDispencer2DoseVolumeCV 	:= eRFID[iw6].lrDoseVolumeCV;	//Do wykresów HMI
								IF eRFID[iw6].nDispencerNr = 1 THEN
									VIS.lrDispencer1DoseVolumeCV :=	eRFID[iw6].lrDoseVolumeCV;	
								ELSIF eRFID[iw6].nDispencerNr = 2 THEN
									VIS.lrDispencer2DoseVolumeCV :=	eRFID[iw6].lrDoseVolumeCV;
								ELSIF eRFID[iw6].nDispencerNr = 3 THEN
									VIS.lrDispencer3DoseVolumeCV :=	eRFID[iw6].lrDoseVolumeCVSecondPhase;							
								ELSIF eRFID[iw6].nDispencerNr = 4 THEN
									VIS.lrDispencer4DoseVolumeCV :=	eRFID[iw6].lrDoseVolumeCVSecondPhase;	
								ELSE									  
									VIS.lrDispencer4DoseVolumeCV := 0.0;
								END_IF	
							
								(*IF eRFID[iw6].nDispencerNr = 1 THEN
									VIS.lrDispencer1WeightMeasured := eRFID[iw6].lrWeightCV;	//Do wykresów HMI
									VIS.lrDispencer1DoseVolumeCV :=	eRFID[iw6].lrDoseVolumeCV;	//Do wykresów HMI
									VIS.bDispencer1WeightMeasured := TRUE; //Do wyświetlenia na ekranie głównym
								ELSE									  
									VIS.lrDispencer1WeightMeasured := VIS.lrDispencer1DoseVolumeCV := 0.0;	//Do wykresów HMI
									VIS.bDispencer1WeightMeasured := FALSE; //Do wyświetlenia na ekranie głównym
								END_IF
								IF eRFID[iw6].nDispencerNr = 2 THEN
									VIS.lrDispencer2WeightMeasured := eRFID[iw6].lrWeightCV;	//Do wykresów HMI
									VIS.lrDispencer2DoseVolumeCV :=	eRFID[iw6].lrDoseVolumeCV;	//Do wykresów HMI
									VIS.bDispencer2WeightMeasured := TRUE; //Do wyświetlenia na ekranie głównym
									IF bDosingTwoPhases THEN
										VIS.lrDispencer2DoseVolumeCV :=	eRFID[iw6].lrDoseVolumeCVSecondPhase; //Do wykresów HMI
									END_IF
								ELSE									
									VIS.lrDispencer2WeightMeasured := VIS.lrDispencer2DoseVolumeCV := 0.0;	//Do wykresów HMI
									VIS.bDispencer2WeightMeasured := FALSE; //Do wyświetlenia na ekranie głównym
								END_IF
								IF eRFID[iw5].nDispencerNr = 3 THEN
									VIS.lrDispencer3WeightMeasured := eRFID[iw6].lrWeightCV;	//Do wykresów HMI
									VIS.lrDispencer3DoseVolumeCV :=	eRFID[iw6].lrDoseVolumeCV;	//Do wykresów HMI
									VIS.bDispencer3WeightMeasured := TRUE; //Do wyświetlenia na ekranie głównym
								ELSE									  
									VIS.lrDispencer3WeightMeasured := VIS.lrDispencer3DoseVolumeCV := 0.0;	//Do wykresów HMI
									VIS.bDispencer3WeightMeasured := FALSE; //Do wyświetlenia na ekranie głównym
								END_IF
								
								IF eRFID[iw6].nDispencerNr = 4 THEN
									VIS.lrDispencer4WeightMeasured := eRFID[iw6].lrWeightCV;	//Do wykresów HMI
									VIS.lrDispencer4DoseVolumeCV :=	eRFID[iw6].lrDoseVolumeCV;	//Do wykresów HMI
									VIS.bDispencer4WeightMeasured := TRUE; //Do wyświetlenia na ekranie głównym
								ELSE									  
									VIS.lrDispencer4WeightMeasured := VIS.lrDispencer4DoseVolumeCV := 0.0;	//Do wykresów HMI
									VIS.bDispencer4WeightMeasured := FALSE; //Do wyświetlenia na ekranie głównym
								END_IF*)
								
								(*Koniec generowania danych do wykresów*)
								IF 	((LREAL_TO_DINT(eRFID[iw6].lrWeightCV)-LREAL_TO_DINT(eRFID[iw6].lrWeightSV))<=(lrWeightUpperTolerance)) AND 
									((LREAL_TO_DINT(eRFID[iw6].lrWeightSV)-LREAL_TO_DINT(eRFID[iw6].lrWeightCV))<=lrWeightLowerTolerance) 
									THEN
									eRFID[iw6].bWeightOK := eWeightPackage2PhasePackageState[2].bWeightOK := TRUE;
								END_IF	
								(*Dodatkowa informacja o wadze*)
								IF 	((LREAL_TO_DINT(eRFID[iw6].lrWeightCV)-LREAL_TO_DINT(eRFID[iw6].lrWeightSV))>lrWeightUpperTolerance) THEN
									eRFID[iw6].bWeightTooHigh := eWeightPackage2PhasePackageState[2].bWeightTooHigh := TRUE;
								END_IF
								IF ((LREAL_TO_DINT(eRFID[iw6].lrWeightSV)-LREAL_TO_DINT(eRFID[iw6].lrWeightCV))>lrWeightLowerTolerance) THEN
									eRFID[iw6].bWeightTooLow:= eWeightPackage2PhasePackageState[2].bWeightTooLow := TRUE;
								END_IF

							VIS.bWeight6DoWeighting:=FALSE;
	
							END_IF																		
						ELSIF NOT bWeight1Enable THEN
							eRFID[iw6].bWeightOK := eWeightPackage2PhasePackageState[2].bWeightOK := TRUE;
							eRFID[iw6].bWeightTooHigh := eWeightPackage2PhasePackageState[2].bWeightTooHigh := FALSE;
							eRFID[iw6].bWeightTooLow:= eWeightPackage2PhasePackageState[2].bWeightTooLow := FALSE;
							eRFID[iw6].lrWeightMeasuredCV := eWeightPackage2PhasePackageState[2].lrWeightMeasuredCV := 0;
							eRFID[iw6].lrWeightCV := eWeightPackage2PhasePackageState[2].lrWeightCV :=VIS.lrWeight6Mass:=lrWeightMassSV;	
							eRFID[iw6].lrWeightSV := eWeightPackage2PhasePackageState[2].lrWeightSV :=lrWeightMassSV;
							eRFID[iw6].bWeighed := eWeightPackage2PhasePackageState[2].bWeighed  := FALSE;
						END_IF
						//KONIEC WARUNKI STACJI								
				ELSIF tonWeightPackageState6BnCardNumber0.Q THEN	// Jeżeli nie wykryje RFID
					VIS.bWeight6DoWeighting 					:= FALSE;
					eWeightPackage2PhasePackageState[2].bFormPresent	:= TRUE;	//Dp	
					eWeightPackage2PhasePackageState[2].bWeightOK 	:= FALSE;
					eWeightPackage2PhasePackageState[2].bWeighed 	:= TRUE;
				ELSIF tonWeightPackageState6BnNoCardNumber.Q THEN 	// Jeżeli nie ma RFID w tablicy
					VIS.bWeight6DoWeighting 					:= FALSE;
					eWeightPackage2PhasePackageState[2].bWeightOK 	:= FALSE;
					eWeightPackage2PhasePackageState[2].bWeighed 	:= TRUE;
				ELSE
					;
				END_IF
				
			END_FOR	
		END_IF
END_ACTION

ACTION aP05_WeightBlock:

IF bLidFeederEnable OR bWickFeederEnable THEN
	IF 
	eBeforeLidFeeder2PackageState[4].bFormPresent OR
	eBeforeLidFeeder2PackageState[3].bFormPresent OR
	eBeforeLidFeeder2PackageState[2].bFormPresent //OR
	//eBeforeLidFeeder2PackageState[1].bFormPresent	
	THEN
		bWeight1234ReleaseBlock := TRUE;
	ELSE
		bWeight1234ReleaseBlock := FALSE;
	END_IF

ELSE
	bWeight1234ReleaseBlock :=	FALSE;
END_IF



IF bDosingTwoPhases THEN
	IF ((*MAIN.IbLidSealerAfterSensor OR*) MAIN.IbLidSealerSecondFormSensor OR MAIN.IbLidFeederAfterSensor) AND (P00_PackML.fbPMLAuto.ePMLState = E_PMLState.ePMLState_EXECUTE)
	THEN
		bWeight56ReleaseBlock := TRUE;
	ELSE
		bWeight56ReleaseBlock := FALSE;
	END_IF

ELSE
	bWeight56ReleaseBlock :=	FALSE;
END_IF
END_ACTION

ACTION aP05_WeightGateBefore:
(*
Nazwa:			aP05_WeightGateBefore
Opis:			Szlabany przed wagą
Wersja:			v0.1
Data:			2024-04-09
Autor:			DP
Urzadzenia:		
Konfiguracja:	
Info:
*)
toWeightRealeseByLidFeeder (IN:= 	(	
										(
										NOT P05_Weight.fbIbWeight1FormBeforeSensor.bOUT AND
										NOT P05_Weight.fbIbWeight2FormBeforeSensor.bOUT AND
										NOT P05_Weight.fbIbWeight3FormBeforeSensor.bOUT AND
										NOT P05_Weight.fbIbWeight4FormBeforeSensor.bOUT AND 
										NOT P05_Weight.tonIbWeight1FormSensor.Q
										) OR
										NOT bLidFeederEnable
									), PT := T#50MS);




VIS.bGateBeforeWeight14Run;
VIS.bGateBeforeWeight56Run;
toniWeight14GateBeforeCASE	(IN:=	iWeightGateBeforeCASE = 60, PT:=T#0MS);
tonbGateBeforeWeight14Run	(IN:=	NOT eAfterDispencersPackageState[1].bFormPresent AND 
									NOT eAfterDispencersPackageState[2].bFormPresent AND 
									NOT eAfterDispencersPackageState[3].bFormPresent AND 
									NOT eAfterDispencersPackageState[4].bFormPresent 
									,PT:=T#100MS);
toniWeight14GateBeforeCASE2	(IN:=	iWeightGateBeforeCASE = 50 AND 
									eAfterDispencersPackageState[1].bFormPresent AND 
									eAfterDispencersPackageState[2].bFormPresent AND 
									eAfterDispencersPackageState[3].bFormPresent AND 
									eAfterDispencersPackageState[4].bFormPresent AND 
									VIS.bGateBeforeWeight14Run AND
									NOT eWeightPackageState[1].bFormPresent AND
									NOT eWeightPackageState[2].bFormPresent AND
									NOT eWeightPackageState[3].bFormPresent AND
									NOT eWeightPackageState[4].bFormPresent
									AND
									toWeightRealeseByLidFeeder.Q
									
									
									,PT:= T#10S);
//fbIbWeight14Gate4FormBeforeSensor	(bIN:= NOT P05_Weight.IbWeight4ActuatorSensorUp,	tFilterTimeOn:=T#250MS,	tFilterTimeOff:=T#80MS); //bylo 150 i 80
fbIbWeight14Gate4FormBeforeSensor	(bIN:= (P05_Weight.QbWeight4Actuator AND P05_Weight.IbWeight4FormSensor) OR (NOT P05_Weight.IbWeight4FormSensor (*AND NOT P05_Weight.IbWeight3FormSensor*)),	tFilterTimeOn:=T#300MS,	tFilterTimeOff:=T#80MS); //bylo 150 i 80

											
toniWeight56GateBeforeCASE	(IN:=	iWeightGateBeforeCASE = 60, PT:=T#0MS);
tonbGateBeforeWeight56Run	(IN:=	NOT eAfterDispencer12PackageState2Phase[1].bFormPresent AND 
									NOT eAfterDispencer12PackageState2Phase[2].bFormPresent 
									,PT:=T#100MS);
toniWeight56GateBeforeCASE2	(IN:=	iWeightGateBeforeCASE = 50 AND 
									eAfterDispencer12PackageState2Phase[1].bFormPresent AND 
									eAfterDispencer12PackageState2Phase[2].bFormPresent AND
									VIS.bGateBeforeWeight56Run AND
									NOT eWeightPackage2PhasePackageState[1].bFormPresent AND
									NOT eWeightPackage2PhasePackageState[2].bFormPresent 
									,PT:= T#10S);															
fbIbWeight56Gate6FormBeforeSensor	(bIN:=NOT P05_Weight.IbWeight6ActuatorSensorUp,	tFilterTimeOn:=T#150MS,	tFilterTimeOff:=T#80MS);
IF NOT bEXPACK THEN									
	CASE iWeightGateBeforeCASE OF 
		
		0:
			IF bWeight1Enable THEN
				iWeightGateBeforeCASE			:=	iWeightGateBeforeCASE	+	10;
			ELSE
				VIS.bGateBeforeWeight14Run		:=	FALSE;
				VIS.bGateBeforeWeight56Run		:=	FALSE;			
			END_IF
		10:
			iWeightGateBeforeCASE			:=	iWeightGateBeforeCASE	+	10;
			
		20:
			IF tonLongDelayAfterStart.Q THEN
				IF (NOT  bDosingTwoPhases AND eAfterDispencersPackageState[1].bFormPresent 			AND eAfterDispencersPackageState[2].bFormPresent 		AND eAfterDispencersPackageState[3].bFormPresent AND eAfterDispencersPackageState[4].bFormPresent) OR 
						(bDosingTwoPhases AND eAfterDispencer12PackageState2Phase[1].bFormPresent	AND eAfterDispencer12PackageState2Phase[2].bFormPresent) 
				 THEN
					iWeightGateBeforeCASE		:=	iWeightGateBeforeCASE	+	10;
				END_IF
			END_IF
			
		30:
			IF 	(
					NOT  bDosingTwoPhases AND
					(
					(P05_Weight.eWeightStationRunningState = E_WeightLiftStationState.eReady) OR 
					(P05_Weight.eWeightStationRunningState = E_WeightLiftStationState.eStorageOfForms) OR 
					(P05_Weight.eWeightStationRunningState = E_WeightLiftStationState.eDepartureOfForms) OR 
					(P05_Weight.eWeightStationRunningState = E_WeightLiftStationState.eDisabled 
					)  
					) AND
					NOT P05_Weight.tonIbWeight1ActuatorSensorUp.Q AND 
					NOT P05_Weight.tonIbWeight2ActuatorSensorUp.Q  AND 
					NOT P05_Weight.tonIbWeight3ActuatorSensorUp.Q  AND 
					NOT P05_Weight.tonIbWeight4ActuatorSensorUp.Q  AND
					iFormatOnWeightCounter <= 3 AND 
					NOT (P05_Weight.eWeightStationRunningState = E_WeightLiftStationState.eRepair) AND
					//(VIS.iNumbersOfFormsBetweenWeightAndScrewers <= P00_PackML.iSetNumbersOfFormsBetweenWeightAndScrewers OR VIS.bWeight1EnableShow) AND
					(NOT fbIbCapSorterGateWeightSensor.bOUT OR VIS.bWeight1EnableShow) AND
					toWeightRealeseByLidFeeder.Q
					
				)
				OR
				(
				 	bDosingTwoPhases AND
					(
					(P05_Weight.eWeightStation2PhaseRunningState = E_WeightLiftStationState.eReady) OR 
					(P05_Weight.eWeightStation2PhaseRunningState = E_WeightLiftStationState.eStorageOfForms) OR 
					(P05_Weight.eWeightStation2PhaseRunningState = E_WeightLiftStationState.eDepartureOfForms) OR 
					(P05_Weight.eWeightStation2PhaseRunningState = E_WeightLiftStationState.eDisabled)  
					) AND
					NOT P05_Weight.tonIbWeight5ActuatorSensorUp.Q AND 
					NOT P05_Weight.tonIbWeight6ActuatorSensorUp.Q   AND
					iFormatOnWeightCounter <= 3 AND 
					NOT (P05_Weight.eWeightStation2PhaseRunningState = E_WeightLiftStationState.eRepair) AND
					//(VIS.iNumbersOfFormsBetweenWeightAndScrewers <= P00_PackML.iSetNumbersOfFormsBetweenWeightAndScrewers OR VIS.bWeight1EnableShow)
					(NOT fbIbCapSorterGateWeightSensor.bOUT OR VIS.bWeight1EnableShow)
				) 		
				
			THEN
				//iWeightGateBeforeCASE		:=	iWeightGateBeforeCASE	+	10;
				iWeightGateBeforeCASE		:=	iWeightGateBeforeCASE	+	5;
			END_IF
			
		35: //AutoTara
				//IF VIS.bGateBeforeWeight14Run OR VIS.bGateBeforeWeight56Run THEN
				//	IF bWeighingAutoTarePreset THEN
				//		bWeighingAutoTarePreset 	:=	FALSE;
				//		bWeighingAutoTare			:=	TRUE;
				//	END_IF
				//	IF NOT bWeighingAutoTare OR (P00_PackML.fbPMLAuto.ePMLState = E_PMLState.ePMLState_STOPPING) THEN
				//		iWeightGateBeforeCASE		:=	iWeightGateBeforeCASE	+	5;
				//	END_IF
				//ELSE
					iWeightGateBeforeCASE		:=	iWeightGateBeforeCASE	+	5;
				//END_IF
		40:
			IF NOT (P00_PackML.fbPMLAuto.ePMLState = E_PMLState.ePMLState_STOPPING) THEN
				VIS.bGateBeforeWeight14Run		:=	FALSE;
				VIS.bGateBeforeWeight56Run		:=	FALSE;			
				iWeightGateBeforeCASE			:=	iWeightGateBeforeCASE	+	10;
			END_IF
			
		50:
			IF (
				NOT  bDosingTwoPhases AND
				(P05_Weight.eWeightStationRunningState = E_WeightLiftStationState.eWeighingCycleON OR NOT bWeight1Enable OR toniWeight14GateBeforeCASE2.Q) AND 
				fbIbWeight14Gate4FormBeforeSensor.bOut
				)	//ina czasowka wieksza
				OR 
				(bDosingTwoPhases AND
				(P05_Weight.eWeightStation2PhaseRunningState = E_WeightLiftStationState.eWeighingCycleON OR NOT bWeight1Enable  OR toniWeight56GateBeforeCASE2.Q) AND 
				fbIbWeight56Gate6FormBeforeSensor.bOut)
			THEN
				iWeightGateBeforeCASE		:=	iWeightGateBeforeCASE	+	10;
			END_IF
	 
			IF 
				(NOT  bDosingTwoPhases AND
				tonbGateBeforeWeight14Run.Q AND
				fbIbWeight14Gate4FormBeforeSensor.bOut	
				) 		
			THEN
				VIS.bGateBeforeWeight14Run		:=	TRUE;
			END_IF
			IF 
				(bDosingTwoPhases AND
				tonbGateBeforeWeight56Run.Q AND
				fbIbWeight56Gate6FormBeforeSensor.bOut
				) 			
			THEN
				VIS.bGateBeforeWeight56Run		:=	TRUE;
			END_IF
			
		60:
			IF NOT bDosingTwoPhases THEN
				VIS.bGateBeforeWeight14Run		:=	TRUE;
			ELSIF bDosingTwoPhases THEN
				VIS.bGateBeforeWeight56Run		:=	TRUE;
			END_IF
			IF (NOT bDosingTwoPhases AND 
				toniWeight14GateBeforeCASE.Q) OR
				(bDosingTwoPhases AND 
				toniWeight56GateBeforeCASE.Q) 
				 THEN
					iWeightGateBeforeCASE		:=	0;
			END_IF
			
	END_CASE
ELSE
		CASE iWeightGateBeforeCASE OF 
		
		0:
			IF bWeight1Enable OR (VIS.bDosingTwoPhasesShow AND P05_Weight.IbWeight6FormSensor AND NOT MAIN.IbSecondFormCheckFormSensor) THEN
				iWeightGateBeforeCASE			:=	iWeightGateBeforeCASE	+	10;
			ELSE
				VIS.bGateBeforeWeight14Run		:=	FALSE;
				VIS.bGateBeforeWeight56Run		:=	FALSE;			
			END_IF
		10:
			iWeightGateBeforeCASE			:=	iWeightGateBeforeCASE	+	10;
			
		20:
			IF tonLongDelayAfterStart.Q THEN
				IF (NOT  bDosingTwoPhases AND eAfterDispencersPackageState[1].bFormPresent 			AND eAfterDispencersPackageState[2].bFormPresent 		AND eAfterDispencersPackageState[3].bFormPresent AND eAfterDispencersPackageState[4].bFormPresent) OR 
						(bDosingTwoPhases AND eAfterDispencer12PackageState2Phase[1].bFormPresent	AND eAfterDispencer12PackageState2Phase[2].bFormPresent) 
				 THEN
					iWeightGateBeforeCASE		:=	iWeightGateBeforeCASE	+	10;
				END_IF
			END_IF
			
		30:
			IF 	(
					NOT  bDosingTwoPhases AND
					(
					(P05_Weight.eWeightStationRunningState = E_WeightLiftStationState.eReady) OR 
					(P05_Weight.eWeightStationRunningState = E_WeightLiftStationState.eStorageOfForms) OR 
					(P05_Weight.eWeightStationRunningState = E_WeightLiftStationState.eDepartureOfForms) OR 
					(P05_Weight.eWeightStationRunningState = E_WeightLiftStationState.eDisabled 
					)  
					) AND
					NOT P05_Weight.tonIbWeight1ActuatorSensorUp.Q AND 
					NOT P05_Weight.tonIbWeight2ActuatorSensorUp.Q  AND 
					NOT P05_Weight.tonIbWeight3ActuatorSensorUp.Q  AND 
					NOT P05_Weight.tonIbWeight4ActuatorSensorUp.Q  AND
					iFormatOnWeightCounter <= 3 AND 
					NOT (P05_Weight.eWeightStationRunningState = E_WeightLiftStationState.eRepair) AND
					//(VIS.iNumbersOfFormsBetweenWeightAndScrewers <= P00_PackML.iSetNumbersOfFormsBetweenWeightAndScrewers OR VIS.bWeight1EnableShow) AND
					(NOT fbIbCapSorterGateWeightSensor.bOUT OR VIS.bWeight1EnableShow) AND
					toWeightRealeseByLidFeeder.Q
					
				)
				OR
				(
				 	bDosingTwoPhases AND
					(
					(P05_Weight.eWeightStation2PhaseRunningState = E_WeightLiftStationState.eReady) OR 
					(P05_Weight.eWeightStation2PhaseRunningState = E_WeightLiftStationState.eStorageOfForms) OR 
					(P05_Weight.eWeightStation2PhaseRunningState = E_WeightLiftStationState.eDepartureOfForms) OR 
					(P05_Weight.eWeightStation2PhaseRunningState = E_WeightLiftStationState.eDisabled)  
					) AND
					NOT P05_Weight.tonIbWeight5ActuatorSensorUp.Q AND 
					NOT P05_Weight.tonIbWeight6ActuatorSensorUp.Q   AND
					iFormatOnWeightCounter <= 3 AND 
					NOT (P05_Weight.eWeightStation2PhaseRunningState = E_WeightLiftStationState.eRepair) 
					//(VIS.iNumbersOfFormsBetweenWeightAndScrewers <= P00_PackML.iSetNumbersOfFormsBetweenWeightAndScrewers OR VIS.bWeight1EnableShow)
					(*NOT fbIbCapSorterGateWeightSensor.bOUT OR VIS.bWeight1EnableShow*)
				) 		
				
			THEN
				//iWeightGateBeforeCASE		:=	iWeightGateBeforeCASE	+	10;
				iWeightGateBeforeCASE		:=	iWeightGateBeforeCASE	+	5;
			END_IF
			
		35: //AutoTara
				//IF VIS.bGateBeforeWeight14Run OR VIS.bGateBeforeWeight56Run THEN
				//	IF bWeighingAutoTarePreset THEN
				//		bWeighingAutoTarePreset 	:=	FALSE;
				//		bWeighingAutoTare			:=	TRUE;
				//	END_IF
				//	IF NOT bWeighingAutoTare OR (P00_PackML.fbPMLAuto.ePMLState = E_PMLState.ePMLState_STOPPING) THEN
				//		iWeightGateBeforeCASE		:=	iWeightGateBeforeCASE	+	5;
				//	END_IF
				//ELSE
					iWeightGateBeforeCASE		:=	iWeightGateBeforeCASE	+	5;
				//END_IF
		40:
			IF NOT (P00_PackML.fbPMLAuto.ePMLState = E_PMLState.ePMLState_STOPPING) THEN
				VIS.bGateBeforeWeight14Run		:=	FALSE;
				VIS.bGateBeforeWeight56Run		:=	FALSE;			
				iWeightGateBeforeCASE			:=	iWeightGateBeforeCASE	+	10;
			END_IF
			
		50:
			IF (
				NOT  bDosingTwoPhases AND
				(P05_Weight.eWeightStationRunningState = E_WeightLiftStationState.eWeighingCycleON OR NOT bWeight1Enable OR toniWeight14GateBeforeCASE2.Q) AND 
				fbIbWeight14Gate4FormBeforeSensor.bOut
				)	//ina czasowka wieksza
				OR 
				(bDosingTwoPhases AND
				(P05_Weight.eWeightStation2PhaseRunningState = E_WeightLiftStationState.eWeighingCycleON OR NOT bWeight1Enable  OR toniWeight56GateBeforeCASE2.Q) AND 
				fbIbWeight56Gate6FormBeforeSensor.bOut)
			THEN
				iWeightGateBeforeCASE		:=	iWeightGateBeforeCASE	+	10;
			END_IF
	 
			IF 
				(NOT  bDosingTwoPhases AND
				tonbGateBeforeWeight14Run.Q AND
				fbIbWeight14Gate4FormBeforeSensor.bOut	
				) 		
			THEN
				VIS.bGateBeforeWeight14Run		:=	TRUE;
			END_IF
			IF 
				(bDosingTwoPhases AND
				tonbGateBeforeWeight56Run.Q AND
				fbIbWeight56Gate6FormBeforeSensor.bOut
				) 			
			THEN
				VIS.bGateBeforeWeight56Run		:=	TRUE;
			END_IF
			
		60:
			IF NOT bDosingTwoPhases THEN
				VIS.bGateBeforeWeight14Run		:=	TRUE;
			ELSIF bDosingTwoPhases THEN
				VIS.bGateBeforeWeight56Run		:=	TRUE;
			END_IF
			IF (NOT bDosingTwoPhases AND 
				toniWeight14GateBeforeCASE.Q) OR
				(bDosingTwoPhases AND 
				toniWeight56GateBeforeCASE.Q) 
				 THEN
					iWeightGateBeforeCASE		:=	0;
			END_IF
			
	END_CASE	
END_IF
END_ACTION

ACTION aP06_LidFeeder:
GVL.bLidFeederDragingStationPrepareRun;
VIS.bLidFeederDragingStationRun;

VIS.bLidFeeder1PrepareRun;
VIS.bLidFeeder1Run;
VIS.bLidFeeder2PrepareRun;
VIS.bLidFeeder2Run;

(***P06_LidFeeder******)

(*Tony*)
tonAfterLidFeederEmpty						(IN:=	NOT eAfterLidFeederPackageState[1].bFormPresent AND NOT eAfterLidFeederPackageState[2].bFormPresent,	PT:=T#10MS);
fbIbLidFeederAfterSensor					(bIN:=	NOT MAIN.IbLidFeederAfterSensor,tFilterTimeOn:=T#100MS, tFilterTimeOff:=T#100MS, bOUT=> );										
fbIbLidFeederAfterSensorLonger				(bIN:=	NOT MAIN.IbLidFeederAfterSensor,tFilterTimeOn:=T#500MS, tFilterTimeOff:=T#100MS, bOUT=> );			
tonLidFeederThirdFormsSensor				(IN:=	MAIN.IbLidFeederThirdFormSensor, 																		PT:=T#20MS);
fbIbLidFeederThirdFormCheckFormSensor		(bIN:=
													MAIN.IbLidFeederThirdFormSensor								AND
													eBeforeLidFeederPackageState[1].bFormPresent				AND 
													eBeforeLidFeederPackageState[2].bFormPresent,//				AND 
													//eBeforeLidFeeder2PackageState[1].bFormPresent,
													tFilterTimeOn:=T#80MS , tFilterTimeOff:=T#35MS, bOUT=> ); //bylo 80 i 35
tonfbLidFeederDragStationNotbCycleDone		(IN:= NOT P06_LidFeeder.fbLidFeederDragStation.bCycleDone, PT:=T#800MS);							
tofbLidFeederDragingStationPrepareRun		(IN:= P06_LidFeeder.fbLidFeederDragStation.bCycleDone, PT:=T#100MS);
tonLidFeederFirstFormSensorBeforeDrag		(IN:=P06_LidFeeder.IbLidFeederFirstFormSensorBeforeDrag, PT:=T#5S);
bLidFeederReady	:=	(NOT bLidFeederEnable OR (
											P06_LidFeeder.fbLidFeeder.eState = E_Station.eReady OR 
											P06_LidFeeder.fbLidFeeder.eRunningState = E_LidFeederState.ePuttingLid 
												)	
					AND
					NOT P06_LidFeeder.fbLidFeeder.bCycleDone AND										
					NOT P06_LidFeeder.fbLidFeeder.bRun) AND
					
					(NOT bLidFeederEnable OR (
												P06_LidFeeder.fbLidFeeder2.eState = E_Station.eReady OR 
												P06_LidFeeder.fbLidFeeder2.eRunningState = E_LidFeederState.ePuttingLid 
											)	
					AND						
					NOT P06_LidFeeder.fbLidFeeder2.bCycleDone AND																						
					NOT P06_LidFeeder.fbLidFeeder2.bRun) 
					
					AND tonDelayAfterStart.Q;	
tonDelayLid1Putting	(IN:=bLidFeederEnable AND eLidFeederPackageState[1].bBottlePresent AND eLidFeederPackageState[1].bWeightOK AND eLidFeederPackageState[1].nCardNumber > 0 AND iLidFeederCase =2, Pt:=T#200MS); 
tonDelayLid2Putting	(IN:=bLidFeederEnable AND eLidFeederPackageState[2].bBottlePresent AND eLidFeederPackageState[2].bWeightOK AND eLidFeederPackageState[2].nCardNumber > 0 AND iLidFeederCase =2, Pt:=T#200MS); 


IF tonDelayAfterStart.Q AND VIS.bBarrierLidFeederRun AND bLidFeederDragingStationEnable THEN		
												// Jak juz było przełączenie
	IF NOT tonLongDelayAfterStart.Q AND NOT tonLongDelayFirstDragingLidFeeder.Q THEN 	// Najpierw przesuwaj formatki od czujnika
		IF  NOT P06_LidFeeder.fbLidFeederDragStation.bCycleDone AND NOT VIS.bLidFeederDragingStationRun AND (fb2IbLidFeederThirdFormSensor.bOut OR (tonLidFeederFirstFormSensorBeforeDrag.Q AND NOT P00_ReadRFIDCard.IbLidFeederReaderTagPresent)) AND fbIbLidFeederAfterSensor.bOut AND NOT (P00_PackML.fbPMLAuto.ePMLState = E_PMLState.ePMLState_STOPPING) THEN
			VIS.bLidFeederDragingStationRun							:= TRUE;
			bFirstDragingLidFeederAfterRestart1						:= TRUE;
		END_IF
	END_IF
	IF P06_LidFeeder.fbLidFeederDragStation.bCycleDone AND bFirstDragingLidFeederAfterRestart1 THEN
		VIS.bLidFeederDragingStationRun								:= FALSE;
		bFirstDragingLidFeederAfterRestart1							:= FALSE;
	END_IF
	
	//Potem jeszcze dwa razy
	IF NOT tonLongDelayAfterStart.Q AND tonLongDelayFirstDragingLidFeeder.Q THEN
		IF tonfbLidFeederDragStationNotbCycleDone.Q AND NOT VIS.bLidFeederDragingStationRun AND iFirstDragingLidFeederAfterRestart2Count < 3  AND fbIbLidFeederAfterSensor.bOut AND NOT (P00_PackML.fbPMLAuto.ePMLState = E_PMLState.ePMLState_STOPPING) THEN
			VIS.bLidFeederDragingStationRun							:= TRUE;	
			bFirstDragingLidFeederAfterRestart2						:= TRUE;
			iFirstDragingLidFeederAfterRestart2Count				:= iFirstDragingLidFeederAfterRestart2Count	+	1;
		END_IF
	END_IF
	IF P06_LidFeeder.fbLidFeederDragStation.bCycleDone AND bFirstDragingLidFeederAfterRestart2 THEN
		VIS.bLidFeederDragingStationRun							:= FALSE;	
	END_IF
		
END_IF 


	
(**** Rozpoczynanie cyklu ***)
bLidFeederDragDelayAfterStartFullRegister;
IF tonDelayAfterStart.Q AND fb2IbLidFeederThirdFormSensor.bOUT AND NOT bLidFeederDragDelayAfterStartFullRegister THEN
		eBeforeLidFeeder2PackageState[1].bFormPresent	:= TRUE;
		eBeforeLidFeederPackageState[2].bFormPresent	:= TRUE;
		eBeforeLidFeederPackageState[1].bFormPresent	:= TRUE;
		bLidFeederDragDelayAfterStartFullRegister		:= TRUE;
END_IF
	
(**Prepare*)				
IF	bLidFeederDragingStationEnable AND 	tonLongDelayAfterStart.Q AND NOT P06_LidFeeder.fbLidFeederDragStation.bCycleDone AND
								fbIbLidFeederThirdFormCheckFormSensor.bOut AND 
								tonDelayAfterStart.Q AND 
								bLidFeederDragDelayAfterStartFullRegister AND iLidFeederDragCase = 10 AND
								NOT bLidFeederDragingStationPrepareRun AND NOT VIS.bLidFeederDragingStationRun AND
								P06_LidFeeder.fbLidFeederDragStation.eState = E_Station.eReady AND
								NOT tofbLidFeederDragingStationPrepareRun.Q
THEN
	bLidFeederDragingStationPrepareRun	:=	TRUE;
END_IF

IF (P00_PackML.fbPMLAuto.ePMLState = E_PMLState.ePMLState_STOPPING) THEN
	bLidFeederDragingStationPrepareRun	:=	FALSE;
END_IF

(*Drag*)
CASE iLidFeederDragCase OF
	0:
		IF bLidFeederDragingStationEnable AND tonLongDelayAfterStart.Q AND NOT VIS.bLidFeederDragingStationRun AND NOT P06_LidFeeder.fbLidFeederDragStation.bCycleDone AND VIS.bBarrierLidFeederRun AND
			P06_LidFeeder.fbLidFeederDragStation.eState = E_Station.eReady	
		THEN
			iLidFeederDragCase				:=	10;
		END_IF
	//Po staremu	
	10: 
		IF  (eBeforeLidFeederPackageState[1].bFormPresent AND eBeforeLidFeederPackageState[2].bFormPresent AND eBeforeLidFeeder2PackageState[1].bFormPresent) AND
			(eLidFeederPackageState[1].bLidPutted OR eLidFeederPackageState[1].bLidPutAborted OR NOT eLidFeederPackageState[1].bBottlePresent OR NOT eLidFeederPackageState[1].bLidPuttedOK) AND
			(eLidFeederPackageState[2].bLidPutted OR eLidFeederPackageState[2].bLidPutAborted OR NOT eLidFeederPackageState[2].bBottlePresent OR NOT eLidFeederPackageState[2].bLidPuttedOK) AND			
			tonLidFeederThirdFormsSensor.Q AND (bLidFeederReady OR NOT bLidFeederEnable) AND
			bLidFeederDragDelayAfterStartFullRegister AND 
			tonAfterLidFeederEmpty.Q AND
			NOT eAfterLidFeederPackageState[1].bFormPresent AND NOT eAfterLidFeederPackageState[2].bFormPresent AND
			fbIbLidFeederThirdFormCheckFormSensor.bOUT AND 
			iLidFeederDragStoppingCount < 3 AND
			tonDelayAfterStart.Q
		THEN 
			VIS.bLidFeederDragingStationRun	:=	TRUE;
			IF (P00_PackML.fbPMLAuto.ePMLState = E_PMLState.ePMLState_STOPPING)	THEN
				iLidFeederDragStoppingCount	:=	iLidFeederDragStoppingCount	+	1;
			END_IF
			iLidFeederDragCase				:=	20;
		END_IF
	20:
		iLidFeederDragCase:=25;
	//10: 
	//	IF  (eBeforeLidFeederPackageState[1].bFormPresent AND eBeforeLidFeederPackageState[2].bFormPresent AND eBeforeLidFeeder2PackageState[1].bFormPresent) AND
	//		(eLidFeederPackageState[1].bLidPutted OR eLidFeederPackageState[1].bLidPutAborted OR NOT eLidFeederPackageState[1].bBottlePresent OR NOT eLidFeederPackageState[1].bLidPuttedOK) AND
	//		(eLidFeederPackageState[2].bLidPutted OR eLidFeederPackageState[2].bLidPutAborted OR NOT eLidFeederPackageState[2].bBottlePresent OR NOT eLidFeederPackageState[2].bLidPuttedOK) AND			
	//		tonLidFeederThirdFormsSensor.Q AND (bLidFeederReady OR NOT bLidFeederEnable) AND
	//		bLidFeederDragDelayAfterStartFullRegister AND 
	//		tonAfterLidFeederEmpty.Q AND
	//		NOT eAfterLidFeederPackageState[1].bFormPresent AND NOT eAfterLidFeederPackageState[2].bFormPresent AND
	//		fbIbLidFeederThirdFormCheckFormSensor.bOUT AND 
	//		iLidFeederDragStoppingCount < 3 AND
	//		tonDelayAfterStart.Q
	//	THEN 
	//		iLidFeederDragCase				:=	20;
	//	END_IF
	//20:	
	//	IF iLidSealerDragCase=20 THEN
	//		VIS.bLidFeederDragingStationRun	:=	TRUE;
	//		iLidFeederDragCase:=25;
	//	END_IF
	//	IF (P00_PackML.fbPMLAuto.ePMLState = E_PMLState.ePMLState_STOPPING)	THEN
	//		iLidFeederDragStoppingCount	:=	iLidFeederDragStoppingCount	+	1;
	//	END_IF
	25: 
		IF P06_LidFeeder.fbLidFeederDragStation.bCycleDone OR NOT VIS.bLidFeederDragingStationRun THEN
			iLidFeederDragCase:=30;
		END_IF
		//IF NOT VIS.bLidFeederDragingStationRun THEN
		//	iLidFeederDragCase:=0;
		//END_IF
		
	30: // jak skonczylo zakręcanie to wroc do poczatku
		VIS.bLidFeederDragingStationRun					:=	FALSE;
		bLidFeederDragingStationPrepareRun			:=	FALSE;
		iLidFeederDragCase								:=	50;
	50:
		IF iLidFeederDragStoppingCount < 3 THEN
			iLidFeederDragCase:=0;	
		END_IF
END_CASE


(************************************)
//Deklaracja opóźnienia startu zakręcania
tonStartLidFeederDelay();
tonStartLidFeederDelay.IN:=	(P00_PackML.fbPMLAuto.ePMLState = E_PMLState.ePMLState_EXECUTE OR (P00_PackML.fbPMLAuto.ePMLState = E_PMLState.ePMLState_STOPPING AND iLidFeederDragStoppingCount < 3)) AND 
							((eLidFeederPackageState[1].bFormPresent) AND
							(NOT eLidFeederPackageState[1].bLidPutted AND NOT eLidFeederPackageState[1].bLidPutAborted )) AND
							((eLidFeederPackageState[2].bFormPresent) AND 
							(NOT eLidFeederPackageState[2].bLidPutted AND NOT eLidFeederPackageState[2].bLidPutAborted ))
;
tonStartLidFeederDelay.PT:=INT_TO_TIME(200);




IF bLidFeederEnable THEN
	
	IF iLidFeederCase = 1 THEN
		IF 
			bLidFeederEnable AND 
			NOT P06_LidFeeder.fbLidFeeder.bCycleDone AND
			eBeforeLidFeederPackageState[1].bBottlePresent (*AND eLidFeederPackageState[1].bWeightOK*) AND eBeforeLidFeederPackageState[1].nCardNumber > 0  AND
			P06_LidFeeder.fbLidFeeder.eState = E_Station.eReady AND NOT VIS.bLidFeeder1PrepareRun  AND NOT VIS.bLidFeeder1Run
		THEN
			VIS.bLidFeeder1PrepareRun 									:=	TRUE;
		END_IF
		
		IF bLidFeederEnable AND 
			NOT P06_LidFeeder.fbLidFeeder2.bCycleDone AND
			eBeforeLidFeederPackageState[2].bBottlePresent (*AND eLidFeederPackageState[1].bWeightOK*) AND eBeforeLidFeederPackageState[2].nCardNumber > 0  AND
			P06_LidFeeder.fbLidFeeder2.eState = E_Station.eReady AND NOT VIS.bLidFeeder2PrepareRun  AND NOT VIS.bLidFeeder2Run
		THEN
			VIS.bLidFeeder2PrepareRun 									:=	TRUE;
		END_IF
	END_IF
	
	IF 	P00_PackML.fbPMLAuto.ePMLState = E_PMLState.ePMLState_STOPPING THEN
		VIS.bLidFeeder1PrepareRun 									:=	FALSE;
		VIS.bLidFeeder2PrepareRun 									:=	FALSE;
	END_IF

	
	bLidFeederFormPositioningRun :=	P06_LidFeeder.fbLidFeeder.eRunningState = E_LidFeederState.ePuttingLid2		OR P06_LidFeeder.fbLidFeeder.eRunningState = E_LidFeederState.eHeating OR
									P06_LidFeeder.fbLidFeeder2.eRunningState = E_LidFeederState.ePuttingLid2	OR P06_LidFeeder.fbLidFeeder2.eRunningState = E_LidFeederState.eHeating;

	CASE iLidFeederCase OF
		0:
			iLidFeederCase	:= 1;
	
		1: //Wykrywanie podjechania nowych wózków i opóźnienie
			IF	tonStartLidFeederDelay.Q AND tonDelayAfterStart.Q AND VIS.bBarrierLidFeederRun THEN	
				iLidFeederCase	:= 2;
			END_IF
			
		2:	//Rozpoczecie 
			IF (*tonDelayLid1Putting.q AND*) bLidFeederEnable AND eLidFeederPackageState[1].bBottlePresent AND eLidFeederPackageState[1].bWeightOK AND eLidFeederPackageState[1].nCardNumber > 0  
			THEN			
				VIS.bLidFeeder1Run 										:=	TRUE;
			END_IF
				
			IF (*tonDelayLid2Putting.q AND*) bLidFeederEnable AND eLidFeederPackageState[2].bBottlePresent AND eLidFeederPackageState[2].bWeightOK AND eLidFeederPackageState[2].nCardNumber > 0 
			THEN			
				VIS.bLidFeeder2Run 										:=	TRUE;
			END_IF
			iLidFeederCase	:= 3;
			
		3: //Czekanie na koniec 	
			//Warunek przejścia dalej, albo wykonano zakręcanie albo nie było rozkazu zakręcania (np. brak butelki)
			IF (
				VIS.bLidFeeder1Run AND (P06_LidFeeder.fbLidFeeder.bCycleDone OR P06_LidFeeder.fbLidFeeder.bCycleNotDone)
				OR NOT VIS.bLidFeeder1Run
				) 
				AND
				(
				VIS.bLidFeeder2Run AND (P06_LidFeeder.fbLidFeeder2.bCycleDone OR P06_LidFeeder.fbLidFeeder2.bCycleNotDone)
				OR NOT VIS.bLidFeeder2Run
				)
				THEN
					iLidFeederCase	:= 4;
			END_IF
		
		4: //Zapisywanie rejestrów i kasowanie sygnałów

			eLidFeederPackageState[1].tLidPuttingTime 				:=	P06_LidFeeder.fbLidFeeder.tCycleTime;
			eLidFeederPackageState[2].tLidPuttingTime 				:=	P06_LidFeeder.fbLidFeeder2.tCycleTime;		
			
			IF P06_LidFeeder.fbLidFeeder.bCycleDone THEN
				eLidFeederPackageState[1].bLidPutted 				:=	TRUE;
			ELSIF P06_LidFeeder.fbLidFeeder.bCycleNotDone THEN
				eLidFeederPackageState[1].bLidPutted				:=	FALSE;
				eLidFeederPackageState[1].bLidPutAborted			:=	TRUE;
			ELSIF NOT bLidFeederEnable THEN
				eLidFeederPackageState[1].bLidPutted				:=	TRUE;
			ELSE // Jak wyłączona
				eLidFeederPackageState[1].bLidPutted				:=	TRUE; 
				eLidFeederPackageState[1].bLidPutAborted			:=	TRUE;
			END_IF

			IF P06_LidFeeder.fbLidFeeder2.bCycleDone THEN
				eLidFeederPackageState[2].bLidPutted 				:=	TRUE;
			ELSIF P06_LidFeeder.fbLidFeeder2.bCycleNotDone THEN
				eLidFeederPackageState[2].bLidPutted				:=	FALSE;
				eLidFeederPackageState[2].bLidPutAborted			:=	TRUE;
			ELSIF NOT bLidFeederEnable THEN
				eLidFeederPackageState[2].bLidPutted				:=	TRUE;
			ELSE // Jak wyłączona
				eLidFeederPackageState[2].bLidPutted				:=	TRUE; 
				eLidFeederPackageState[2].bLidPutAborted			:=	TRUE;
			END_IF
						
			FOR y:=1 TO 100 DO
				IF  eRFID[y].nCardNumber=eLidFeederPackageState[1].nCardNumber AND eLidFeederPackageState[1].nCardNumber >0 THEN
				 eRFID[y]:=eLidFeederPackageState[1];
				 EXIT;
				 END_IF;
			END_FOR
			 
			FOR z:=1 TO 100 DO
				IF  eRFID[z].nCardNumber=eLidFeederPackageState[2].nCardNumber AND eLidFeederPackageState[2].nCardNumber >0 THEN
					eRFID[z]:=eLidFeederPackageState[2];
				 EXIT;
				END_IF;
			END_FOR 
			 	
			 iLidFeederCase := 5; 
			 
		5: 
			VIS.bLidFeeder1PrepareRun 									:=	FALSE;	
			VIS.bLidFeeder2PrepareRun 									:=	FALSE;		
			VIS.bLidFeeder1Run 											:=	FALSE;	
			VIS.bLidFeeder2Run 											:=	FALSE;
			

			(***Nie wykonuj dalej ruchu gdy wcisnięty stop lub błąd***)
			IF NOT (P00_PackML.fbPMLAuto.ePMLState = E_PMLState.ePMLState_STOPPING) OR iLidFeederDragStoppingCount < 3 THEN
				iLidFeederCase := 0;
			END_IF
			
	END_CASE
ELSIF NOT bWickFeederEnable THEN
	eLidFeederPackageState[1].bLidPutted 				:=	TRUE;
	eLidFeederPackageState[2].bLidPutted 				:=	TRUE;	
	
	FOR y:=1 TO 100 DO
		IF  eRFID[y].nCardNumber=eLidFeederPackageState[1].nCardNumber AND eLidFeederPackageState[1].nCardNumber >0 THEN
			 eRFID[y]:=eLidFeederPackageState[1];
		EXIT;
		END_IF;
	 END_FOR
			 
	FOR z:=1 TO 100 DO
		IF  eRFID[z].nCardNumber=eLidFeederPackageState[2].nCardNumber AND eLidFeederPackageState[2].nCardNumber >0 THEN
			eRFID[z]:=eLidFeederPackageState[2];
		EXIT;
		END_IF;
	END_FOR 
			 
END_IF
END_ACTION

ACTION aP06_LidPuttedCheck:
VIS.bLidPuttedCheckRun;

fbIbLidPuttedCheck1Sensor					(bIN:=	P06_LidPuttedCheck.IbLidPuttedCheck11Sensor AND P06_LidPuttedCheck.IbLidPuttedCheck12Sensor AND P06_LidPuttedCheck.IbLidPuttedCheck13Sensor,		
													tFilterTimeOn:=T#100MS, tFilterTimeOff:=T#100MS, bOUT=> );																					
fbIbLidPuttedCheck2Sensor					(bIN:=	P06_LidPuttedCheck.IbLidPuttedCheck21Sensor AND P06_LidPuttedCheck.IbLidPuttedCheck22Sensor AND P06_LidPuttedCheck.IbLidPuttedCheck23Sensor,		
													tFilterTimeOn:=T#100MS, tFilterTimeOff:=T#100MS, bOUT=> );										

IF bLidPuttedCheckEnable THEN
	IF iLidSealerDragCase	=	20	THEN
		IF fbIbLidPuttedCheck1Sensor.bOut THEN
			eBeforeLidSealerPackageState[1].bLidPuttedOK		:=	TRUE;
			eBeforeLidSealerPackageState[1].bLidPuttedChecked	:=	TRUE;	
		ELSE
			eBeforeLidSealerPackageState[1].bLidPuttedOK		:=	FALSE;
			eBeforeLidSealerPackageState[1].bLidPuttedChecked	:=	TRUE;				
		END_IF
		IF fbIbLidPuttedCheck2Sensor.bOut THEN
			eBeforeLidSealerPackageState[2].bLidPuttedOK		:=	TRUE;
			eBeforeLidSealerPackageState[2].bLidPuttedChecked	:=	TRUE;	
		ELSE
			eBeforeLidSealerPackageState[2].bLidPuttedOK		:=	FALSE;
			eBeforeLidSealerPackageState[2].bLidPuttedChecked	:=	TRUE;				
		END_IF		
	END_IF

ELSE
	eBeforeLidSealerPackageState[2].bLidPuttedOK		:=	TRUE;
	eBeforeLidSealerPackageState[1].bLidPuttedOK		:=	TRUE;
END_IF
END_ACTION

ACTION aP06_LidSealer:

VIS.bLidSealer1Run;
VIS.bLidSealer2Run;

(***P06_LidSealer******)


(************************************)
//Deklaracja opóźnienia startu zakręcania
tonStartLidSealerDelay();
tonStartLidSealerDelay.IN:=	(P00_PackML.fbPMLAuto.ePMLState = E_PMLState.ePMLState_EXECUTE OR (P00_PackML.fbPMLAuto.ePMLState = E_PMLState.ePMLState_STOPPING AND iFirstDragingLidSealerAfterRestart2Count < 3)) AND
							((eLidSealerPackageState[1].bFormPresent) AND
							(NOT eLidSealerPackageState[1].bLidSealed AND NOT eLidSealerPackageState[1].bLidSealingAborted )) AND
							((eLidSealerPackageState[2].bFormPresent) AND 
							(NOT eLidSealerPackageState[2].bLidSealed AND NOT eLidSealerPackageState[2].bLidSealingAborted ))
;
tonStartLidSealerDelay.PT:=INT_TO_TIME(350);

IF bLidSealerEnable THEN
	CASE iLidSealerCase OF
		0:
			iLidSealerCase	:= 1;
	
		1: //Wykrywanie podjechania nowych wózków i opóźnienie
			IF	tonStartLidSealerDelay.Q AND tonDelayAfterStart.Q AND VIS.bBarrierLidFeederRun THEN	
				iLidSealerCase	:= 2;
			END_IF
			
		2:	//Rozpoczecie 
			IF bLidSealerEnable AND eLidSealerPackageState[1].bBottlePresent AND eLidSealerPackageState[1].bLidPuttedOK AND eLidSealerPackageState[1].nCardNumber > 0  
			THEN			
				VIS.bLidSealer1Run 										:=	TRUE;
			END_IF
				
			IF bLidSealerEnable AND eLidSealerPackageState[2].bBottlePresent AND eLidSealerPackageState[2].bLidPuttedOK AND eLidSealerPackageState[2].nCardNumber > 0 
			THEN			
				VIS.bLidSealer2Run 										:=	TRUE;
			END_IF
			iLidSealerCase	:= 3;
			
		3: //Czekanie na koniec 	
			//Warunek przejścia dalej, albo wykonano zakręcanie albo nie było rozkazu zakręcania (np. brak butelki)
			IF (
				VIS.bLidSealer1Run AND (P06_LidSealer.fbLidSealer.bCycleDone OR P06_LidSealer.fbLidSealer.bCycleNotDone)
				OR NOT VIS.bLidSealer1Run
				) 
				AND
				(
				VIS.bLidSealer2Run AND (P06_LidSealer.fbLidSealer2.bCycleDone OR P06_LidSealer.fbLidSealer2.bCycleNotDone)
				OR NOT VIS.bLidSealer2Run
				)
				THEN
					iLidSealerCase	:= 4;
			END_IF
		
		4: //Zapisywanie rejestrów i kasowanie sygnałów

			eLidSealerPackageState[1].tLidSealingTime 				:=	P06_LidSealer.fbLidSealer.tCycleTime;
			eLidSealerPackageState[2].tLidSealingTime 				:=	P06_LidSealer.fbLidSealer2.tCycleTime;		
			
			IF P06_LidSealer.fbLidSealer.bCycleDone THEN
				eLidSealerPackageState[1].bLidSealed 				:=	TRUE;
			ELSIF P06_LidSealer.fbLidSealer.bCycleNotDone THEN
				eLidSealerPackageState[1].bLidSealed				:=	FALSE;
				eLidSealerPackageState[1].bLidSealingAborted		:=	TRUE;
			ELSIF NOT bLidSealerEnable THEN
				eLidSealerPackageState[1].bLidSealed				:=	TRUE;
			ELSE // Jak wyłączona
				eLidSealerPackageState[1].bLidSealed				:=	TRUE; 
				eLidSealerPackageState[1].bLidSealingAborted			:=	TRUE;
			END_IF

			IF P06_LidSealer.fbLidSealer2.bCycleDone THEN
				eLidSealerPackageState[2].bLidSealed 				:=	TRUE;
			ELSIF P06_LidSealer.fbLidSealer2.bCycleNotDone THEN
				eLidSealerPackageState[2].bLidSealed				:=	FALSE;
				eLidSealerPackageState[2].bLidSealingAborted		:=	TRUE;
			ELSIF NOT bLidSealerEnable THEN
				eLidSealerPackageState[2].bLidSealed				:=	TRUE;
			ELSE // Jak wyłączona
				eLidSealerPackageState[2].bLidSealed				:=	TRUE; 
				eLidSealerPackageState[2].bLidSealingAborted		:=	TRUE;
			END_IF
						
			FOR y:=1 TO 100 DO
				IF  eRFID[y].nCardNumber=eLidSealerPackageState[1].nCardNumber AND eLidSealerPackageState[1].nCardNumber >0 THEN
				 eRFID[y]:=eLidSealerPackageState[1];
				 EXIT;
				 END_IF;
			END_FOR
			 
			FOR z:=1 TO 100 DO
				IF  eRFID[z].nCardNumber=eLidSealerPackageState[2].nCardNumber AND eLidSealerPackageState[2].nCardNumber >0 THEN
					eRFID[z]:=eLidSealerPackageState[2];
				 EXIT;
				END_IF;
			END_FOR 
			 	
			 iLidSealerCase := 5; 
			 
		5: 
			VIS.bLidSealer1Run 											:=	FALSE;	
			VIS.bLidSealer2Run 											:=	FALSE;

			(***Nie wykonuj dalej ruchu gdy wcisnięty stop lub błąd***)
			IF NOT (P00_PackML.fbPMLAuto.ePMLState = E_PMLState.ePMLState_STOPPING) OR iFirstDragingLidSealerAfterRestart2Count < 3 THEN
				iLidSealerCase := 0;
			END_IF
			
	END_CASE
ELSE
	eLidSealerPackageState[1].bLidSealed 				:=	TRUE;
	eLidSealerPackageState[2].bLidSealed 				:=	TRUE;	
	
	FOR y:=1 TO 100 DO
		IF  eRFID[y].nCardNumber=eLidSealerPackageState[1].nCardNumber AND eLidSealerPackageState[1].nCardNumber >0 THEN
			 eRFID[y]:=eLidSealerPackageState[1];
		EXIT;
		END_IF;
	 END_FOR
			 
	FOR z:=1 TO 100 DO
		IF  eRFID[z].nCardNumber=eLidSealerPackageState[2].nCardNumber AND eLidSealerPackageState[2].nCardNumber >0 THEN
			eRFID[z]:=eLidSealerPackageState[2];
		EXIT;
		END_IF;
	END_FOR 
			 
END_IF
END_ACTION

ACTION aP06_LidSealerDrag:
VIS.bLidSealerDragingStationRun;
GVL.bLidSealerDragingStationPrepareRun;

VIS.bLidSealer1Run;
VIS.bLidSealer2Run;


(***P06_LidSealer******)

(*Tony*)
fbIbLidSealerAfterSensor					(bIN:=	NOT MAIN.IbLidSealerAfterSensor,																		tFilterTimeOn:=T#200MS, tFilterTimeOff:=T#150MS, bOUT=> );										

tonLidSealerThirdFormsSensor				(IN:=	MAIN.IbLidSealerSecondFormSensor, 	PT:=T#20MS);

tonLidSealerFirstFormsSensor				(IN:=	MAIN.IbLidSealerFirstFormSensor, 	PT:=T#20MS);
fbIbLidSealerThirdFormCheckFormSensor		(bIN:=
													MAIN.IbLidSealerSecondFormSensor	AND
													eBeforeLidSealerPackageState[1].bFormPresent					AND 
													eBeforeLidSealerPackageState[2].bFormPresent,					
													tFilterTimeOn:=T#50MS , tFilterTimeOff:=T#35MS, bOUT=> ); 
tonfbLidSealerDragStationNotbCycleDone		(IN:= NOT P06_LidSealer.fbLidSealerDragStation.bCycleDone, PT:=T#800MS);												
bLidSealerReady	:=	(NOT bLidSealerEnable OR P06_LidSealer.fbLidSealer.eState = E_Station.eReady AND NOT P06_LidSealer.fbLidSealer.bRun) AND
					(NOT bLidSealerEnable OR P06_LidSealer.fbLidSealer.eState = E_Station.eReady AND NOT P06_LidSealer.fbLidSealer.bRun) 
					AND tonDelayAfterStart.Q;	
tofbLidSealerDragingStationPrepareRun		(IN:= P06_LidSealer.fbLidSealerDragStation.bCycleDone, PT:=T#700MS);

IF bLidSealerDragingStationEnable AND VIS.bBarrierLidFeederRun THEN
//IF VIS.bBarrierLidFeederRun THEN		
												// Jak juz było przełączenie
	IF NOT tonLongDelayAfterStart.Q AND NOT tonLongDelayFirstDragingLidSealer.Q THEN 	// Najpierw przesuwaj formatki od czujnika
		IF  NOT P06_LidSealer.fbLidSealerDragStation.bCycleDone AND NOT VIS.bLidSealerDragingStationRun AND fb2IbLidSealerSecondFormSensor.bOut AND fbIbLidSealerAfterSensor.bOut THEN
			VIS.bLidSealerDragingStationRun							:= TRUE;
			bFirstDragingLidSealerAfterRestart1						:= TRUE;
		END_IF
	END_IF
	IF P06_LidSealer.fbLidSealerDragStation.bCycleDone AND bFirstDragingLidSealerAfterRestart1 THEN
		VIS.bLidSealerDragingStationRun								:= FALSE;
		bFirstDragingLidSealerAfterRestart1							:= FALSE;
	END_IF
	
	//Potem jeszcze dwa razy
	IF NOT tonLongDelayAfterStart.Q AND tonLongDelayFirstDragingLidSealer.Q THEN
		IF tonfbLidSealerDragStationNotbCycleDone.Q AND NOT VIS.bLidSealerDragingStationRun AND iFirstDragingLidSealerAfterRestart2Count < 3 AND fbIbLidSealerAfterSensor.bOut THEN
			VIS.bLidSealerDragingStationRun							:= TRUE;	
			bFirstDragingLidSealerAfterRestart2						:= TRUE;
			iFirstDragingLidSealerAfterRestart2Count				:= iFirstDragingLidSealerAfterRestart2Count	+	1;
		END_IF
	END_IF
	IF P06_LidSealer.fbLidSealerDragStation.bCycleDone AND bFirstDragingLidSealerAfterRestart2 THEN
		VIS.bLidSealerDragingStationRun								:= FALSE;	
	END_IF
		
END_IF 	

		
(**** Rozpoczynanie cyklu ***)
bLidSealerDragDelayAfterStartFullRegister;
IF tonDelayAfterStart.Q AND fb2IbLidSealerSecondFormSensor.bOUT AND NOT bLidSealerDragDelayAfterStartFullRegister THEN
		eBeforeLidSealerPackageState[2].bFormPresent	:= TRUE;
		eBeforeLidSealerPackageState[1].bFormPresent	:= TRUE;
		bLidSealerDragDelayAfterStartFullRegister		:= TRUE;
END_IF
	
(**Prepare*)				
IF	bLidSealerDragingStationEnable AND tonLongDelayAfterStart.Q AND NOT P06_LidSealer.fbLidSealerDragStation.bCycleDone AND
								fbIbLidSealerThirdFormCheckFormSensor.bOut AND
								tonDelayAfterStart.Q AND 
								bLidSealerDragDelayAfterStartFullRegister AND iLidSealerDragCase = 10 AND
								NOT bLidSealerDragingStationPrepareRun  AND NOT  VIS.bLidSealerDragingStationRun AND
								P06_LidSealer.fbLidSealerDragStation.eState = E_Station.eReady AND
								NOT tofbLidSealerDragingStationPrepareRun.Q
THEN
	bLidSealerDragingStationPrepareRun	:=	TRUE;
END_IF

IF (P00_PackML.fbPMLAuto.ePMLState = E_PMLState.ePMLState_STOPPING) THEN
	bLidSealerDragingStationPrepareRun	:=	FALSE;
END_IF

//bLidSelaerDragIfNot2PucksAnd5s
tonLidSelaerDragIfNot2PucksAnd5s	(IN:=
		P00_PackML.fbPMLAuto.ePMLState = E_PMLState.ePMLState_EXECUTE AND
		(P06_LidSealer.fbLidSealerDragStation.eState = E_Station.eReady	 OR P06_LidSealer.fbLidSealerDragStation.eRunningState = E_DragStationState.eLifting) AND	
		tonLidSealerFirstFormsSensor.Q AND 
		fbNotIbLidSealerSecondFormSensor.bOut AND
		NOT MAIN.IbLidFeederAfterSensor AND
		fbIbLidSealerAfterSensor.bOut 
		, PT:=T#1S000MS);	
IF (tonLidSelaerDragIfNot2PucksAnd5s.Q OR bLidSelaerDragIfNot2PucksAnd5s) THEN
		bLidSelaerDragIfNot2PucksAnd5s							:= TRUE;
		VIS.bLidSealerDragingStationRun							:= TRUE; 
	IF P06_LidSealer.fbLidSealerDragStation.bCycleDone THEN
		VIS.bLidSealerDragingStationRun							:= FALSE;
		GVL.bLidSealerDragingStationPrepareRun					:= FALSE;
		bLidSelaerDragIfNot2PucksAnd5s							:= FALSE;	
		eBeforeLidSealerPackageState[2].bFormPresent			:= FALSE;
		eBeforeLidSealerPackageState[1].bFormPresent			:= FALSE;
	END_IF
END_IF
//Koniec bLidSelaerDragIfNot2PucksAnd5s

(*Drag*)
CASE iLidSealerDragCase OF
	0:
		IF bLidSealerDragingStationEnable AND tonLongDelayAfterStart.Q AND NOT VIS.bLidSealerDragingStationRun AND NOT P06_LidSealer.fbLidSealerDragStation.bCycleDone AND	VIS.bBarrierLidFeederRun AND
			P06_LidSealer.fbLidSealerDragStation.eState = E_Station.eReady		
		THEN
			iLidSealerDragCase				:=	10;
		END_IF
	//po staremu	
	10: 
		IF  (eBeforeLidSealerPackageState[1].bFormPresent AND eBeforeLidSealerPackageState[2].bFormPresent) AND
			(eLidSealerPackageState[1].bLidSealed OR eLidSealerPackageState[1].bLidSealingAborted OR NOT eLidSealerPackageState[1].bBottlePresent) AND
			(eLidSealerPackageState[2].bLidSealed OR eLidSealerPackageState[2].bLidSealingAborted OR NOT eLidSealerPackageState[2].bBottlePresent) AND			
		
			tonLidSealerThirdFormsSensor.Q AND (bLidSealerReady OR NOT bLidSealerEnable) AND
			bLidSealerDragDelayAfterStartFullRegister AND 
			fbIbLidSealerAfterSensor.bOUT AND 
			fbIbLidSealerThirdFormCheckFormSensor.bOUT AND 
			tonbFormTransportersScrewerCmdStart.Q AND
			iLidSealerDragStoppingCount < 3 AND
			tonDelayAfterStart.Q AND
			tonLidSealerFirstFormsSensor.Q
		THEN 
			VIS.bLidSealerDragingStationRun			:=	TRUE;
			IF (P00_PackML.fbPMLAuto.ePMLState = E_PMLState.ePMLState_STOPPING)	THEN
				iLidSealerDragStoppingCount	:=	iLidSealerDragStoppingCount	+	1;
			END_IF
			iLidSealerDragCase						:=	20;
		END_IF
	20:
		iLidSealerDragCase:=25;
	//10: 
	//	IF  (eBeforeLidSealerPackageState[1].bFormPresent AND eBeforeLidSealerPackageState[2].bFormPresent AND eBeforeLidSealerPackageState[1].bFormPresent) AND
	//		(eLidSealerPackageState[1].bLidSealed OR eLidSealerPackageState[1].bLidSealingAborted OR NOT eLidSealerPackageState[1].bBottlePresent) AND
	//		(eLidSealerPackageState[2].bLidSealed OR eLidSealerPackageState[2].bLidSealingAborted OR NOT eLidSealerPackageState[2].bBottlePresent) AND			
	//	
	//		tonLidSealerThirdFormsSensor.Q AND (bLidSealerReady OR NOT bLidSealerEnable) AND
	//		bLidSealerDragDelayAfterStartFullRegister AND 
	//		fbIbLidSealerAfterSensor.bOUT AND 
	//		fbIbLidSealerThirdFormCheckFormSensor.bOUT AND 
	//		tonbFormTransportersScrewerCmdStart.Q AND
	//		iLidSealerDragStoppingCount < 3 AND
	//		tonDelayAfterStart.Q AND
	//		tonLidSealerFirstFormsSensor.Q
	//	THEN 
	//		iLidSealerDragCase						:=	20;
	//	END_IF
	//20:	
	//	IF iLidFeederDragCase=20 THEN
	//		VIS.bLidSealerDragingStationRun			:=	TRUE;
	//		iLidSealerDragCase:=25;
	//	END_IF
	//	IF (P00_PackML.fbPMLAuto.ePMLState = E_PMLState.ePMLState_STOPPING)	THEN
	//		iLidSealerDragStoppingCount	:=	iLidSealerDragStoppingCount	+	1;
	//	END_IF
	//	
	25: 
		IF P06_LidSealer.fbLidSealerDragStation.bCycleDone OR NOT VIS.bLidSealerDragingStationRun THEN
			iLidSealerDragCase:=30;
		END_IF
		//IF NOT VIS.bLidSealerDragingStationRun THEN
		//	iLidSealerDragCase:=0;
		//END_IF
		
	30: // jak skonczylo zakręcanie to wroc do poczatku
		VIS.bLidSealerDragingStationRun				:=	FALSE;
		bLidSealerDragingStationPrepareRun			:=	FALSE;
		iLidSealerDragCase							:=	50;
	50:
		IF iLidSealerDragStoppingCount < 3 THEN
			iLidSealerDragCase:=0;	
		END_IF
END_CASE
END_ACTION

ACTION aP06_LidSealerDrag2Phase:
(***aP06_LidSealerDrag2Phase******)

fbIbLidSealerAfterSensor				(bIN:=	NOT MAIN.IbLidSealerAfterSensor,			tFilterTimeOn:=T#100MS, tFilterTimeOff:=T#100MS, bOUT=> ); 
fbIbLidSealerAfterSensor2				(bIN:=	
												NOT MAIN.IbLidFeederThirdFormSensor	AND
												NOT P05_Weight.IbWeight1FormSensor	AND
												NOT P05_Weight.IbWeight2FormSensor	AND											
												NOT P05_Weight.IbWeight3FormSensor	AND											
												NOT P05_Weight.IbWeight4FormSensor											

										,tFilterTimeOn:=T#3S500MS, tFilterTimeOff:=T#0S, bOUT=> );										
											
tonLidSealerDragSecondFormSensor		(IN:=	MAIN.IbLidSealerSecondFormSensor AND MAIN.IbLidSealerFirstFormSensor (*AND (iLidSealerDragFormCounter >= 2)*), 			PT:=T#100MS); //bylo 800

										
(**** Rozpoczynanie cyklu ***)
bLidSealerDragDelayAfterStartFullRegister;
IF (*tonDelayAfterStart.Q AND*) tonLidSealerDragSecondFormSensor.Q AND NOT bLidSealerDragDelayAfterStartFullRegister THEN
	bLidSealerDragDelayAfterStartFullRegister		:= TRUE;
END_IF
			
	
IF (P00_PackML.fbPMLAuto.ePMLState = E_PMLState.ePMLState_STOPPING) THEN
	GVL.bLidSealerDragingStationPrepareRun:=FALSE;
END_IF


CASE iLidSealerDragCase OF
	
	0:
		IF GVL.bLidSealerDragingStationEnable THEN
			iLidSealerDragCase				:=	10;
		END_IF
		
	10: //Sprawdzanie czy są formatki przed 
		IF  
			tonLidSealerDragSecondFormSensor.Q AND 
			bLidSealerDragDelayAfterStartFullRegister AND
			NOT MAIN.IbLidSealerAfterSensor AND 
			fbIbLidSealerAfterSensor.bOUT AND 
			(*fbIbLidSealerAfterSensor2.bOUT AND*)
			tonbFormTransportersScrewerCmdStart.Q AND
			NOT (P00_PackML.fbPMLAuto.ePMLState = E_PMLState.ePMLState_STOPPING) 

		THEN 
			VIS.bLidSealerDragingStationRun			:=	TRUE;
			iLidSealerDragFormCounter				:= 	0;			
			iLidSealerDragCase						:=	20;
		END_IF
		
	20://czy pusto
			iLidSealerDragCase:=25;		
	25: 
		// Reset cyklu jak skonczylo przeciaganie
		IF P06_LidSealer.fbLidSealerDragStation.bCycleDone THEN
			iLidSealerDragCase:=30;
		END_IF
		
		IF NOT VIS.bLidSealerDragingStationRun THEN
			iLidSealerDragCase:=0;
		END_IF
		
	30: // jak skonczylo zakręcanie to wroc do poczatku
		VIS.bLidSealerDragingStationRun				:=	FALSE;
		GVL.bLidSealerDragingStationPrepareRun		:=	FALSE;
		iLidSealerDragCase							:=	50;
		
	50:
		IF NOT (P00_PackML.fbPMLAuto.ePMLState = E_PMLState.ePMLState_STOPPING) THEN
			iLidSealerDragCase:=0;	
		END_IF
END_CASE
END_ACTION

ACTION aP06_WickFeeder:
(*
Nazwa:			aP06_WickFeeder
Opis:			Cykl knotów i przeciągania pod knotami
Wersja:			v0.1
Data:			2025-12-01
Autor:			
Urzadzenia:		
Konfiguracja:	
Info:
*)

GVL.bWickFeederDragingStationPrepareRun;
VIS.bWickFeederDragingStationRun;

VIS.bWickFeederSorterRun;
VIS.bWickFeeder1Run;
VIS.bWickFeeder2Run;

(***P06_WickFeeder******)
(*Tony*)
tonAfterWickFeederEmpty						(IN:=	NOT eAfterLidFeederPackageState[1].bFormPresent AND NOT eAfterLidFeederPackageState[2].bFormPresent,	PT:=T#10MS);
fbIbWickFeederAfterSensor					(bIN:=	NOT MAIN.IbLidFeederAfterSensor,tFilterTimeOn:=T#100MS, tFilterTimeOff:=T#100MS, bOUT=> );										
fbIbWickFeederAfterSensorLonger				(bIN:=	NOT MAIN.IbLidFeederAfterSensor,tFilterTimeOn:=T#500MS, tFilterTimeOff:=T#100MS, bOUT=> );			
tonWickFeederThirdFormsSensor				(IN:=	MAIN.IbLidFeederThirdFormSensor, 																		PT:=T#20MS);
fbIbWickFeederThirdFormCheckFormSensor		(bIN:=
													MAIN.IbLidFeederThirdFormSensor								AND
													eBeforeLidFeederPackageState[1].bFormPresent				AND 
													eBeforeLidFeederPackageState[2].bFormPresent				AND 
													eBeforeLidFeeder2PackageState[1].bFormPresent,
													tFilterTimeOn:=T#80MS , tFilterTimeOff:=T#35MS, bOUT=> ); 
tonfbWickFeederDragStationNotbCycleDone		(IN:= NOT P06_WickFeeder.fbWickFeederDragStation.bCycleDone, PT:=T#800MS);							
tofbWickFeederDragingStationPrepareRun		(IN:= P06_WickFeeder.fbWickFeederDragStation.bCycleDone, PT:=T#100MS);
tonWickFeederFirstFormSensorBeforeDrag		(IN:=P06_LidFeeder.IbLidFeederFirstFormSensorBeforeDrag, PT:=T#5S);
bWickFeederReady	:=	(NOT bWickFeederEnable OR (
											P06_WickFeeder.fbWickFeederSt.eRunningState1 = E_WickFeederState.eReady AND P06_WickFeeder.fbWickFeederSt.eRunningState2 = E_WickFeederState.eReady)	
					AND
					NOT P06_WickFeeder.fbWickFeederSt.bCycleDone1 AND NOT P06_WickFeeder.fbWickFeederSt.bCycleDone2 AND											
					NOT P06_WickFeeder.fbWickFeederSt.bRun1 AND NOT P06_WickFeeder.fbWickFeederSt.bRun2) 

					
					AND tonDelayAfterStart.Q;	
tonDelayWick1Putting	(IN:=bWickFeederEnable AND eLidFeederPackageState[1].bBottlePresent AND eLidFeederPackageState[1].bWeightOK AND eLidFeederPackageState[1].nCardNumber > 0 AND iLidFeederCase =2, Pt:=T#200MS); 
tonDelayWick2Putting	(IN:=bWickFeederEnable AND eLidFeederPackageState[2].bBottlePresent AND eLidFeederPackageState[2].bWeightOK AND eLidFeederPackageState[2].nCardNumber > 0 AND iLidFeederCase =2, Pt:=T#200MS); 


IF tonDelayAfterStart.Q AND VIS.bBarrierLidFeederRun AND bWickFeederDragingStationEnable THEN		
				
	IF NOT tonLongDelayAfterStart.Q AND NOT tonLongDelayFirstDragingLidFeeder.Q THEN 	// Najpierw przesuwaj formatki od czujnika
		IF  NOT P06_WickFeeder.fbWickFeederDragStation.bCycleDone AND NOT VIS.bWickFeederDragingStationRun AND (fb2IbLidFeederThirdFormSensor.bOut OR (tonWickFeederFirstFormSensorBeforeDrag.Q AND NOT P00_ReadRFIDCard.IbLidFeederReaderTagPresent)) AND fbIbWickFeederAfterSensor.bOut AND NOT (P00_PackML.fbPMLAuto.ePMLState = E_PMLState.ePMLState_STOPPING) THEN
			VIS.bWickFeederDragingStationRun							:= TRUE;
			bFirstDragingWickFeederAfterRestart1						:= TRUE;
		END_IF
	END_IF
	IF P06_WickFeeder.fbWickFeederDragStation.bCycleDone AND bFirstDragingWickFeederAfterRestart1 THEN
		VIS.bWickFeederDragingStationRun								:= FALSE;
		bFirstDragingWickFeederAfterRestart1							:= FALSE;
	END_IF
	
	//Potem jeszcze dwa razy
	IF NOT tonLongDelayAfterStart.Q AND tonLongDelayFirstDragingLidFeeder.Q THEN
		IF tonfbWickFeederDragStationNotbCycleDone.Q AND NOT VIS.bWickFeederDragingStationRun AND iFirstDragingWickFeederAfterRestart2Count < 3  AND fbIbWickFeederAfterSensor.bOut AND NOT (P00_PackML.fbPMLAuto.ePMLState = E_PMLState.ePMLState_STOPPING) THEN
			VIS.bWickFeederDragingStationRun							:= TRUE;	
			bFirstDragingWickFeederAfterRestart2						:= TRUE;
			iFirstDragingWickFeederAfterRestart2Count					:= iFirstDragingWickFeederAfterRestart2Count	+	1;
		END_IF
	END_IF
	IF P06_WickFeeder.fbWickFeederDragStation.bCycleDone AND bFirstDragingWickFeederAfterRestart2 THEN
		VIS.bWickFeederDragingStationRun							:= FALSE;	
	END_IF
		
END_IF 


	
(**** Rozpoczynanie cyklu ***)
bWickFeederDragDelayAfterStartFullRegister;
IF tonDelayAfterStart.Q AND fb2IbLidFeederThirdFormSensor.bOUT AND NOT bWickFeederDragDelayAfterStartFullRegister THEN
		//eBeforeLidFeeder2PackageState[1].bFormPresent	:= TRUE; //ok
		eBeforeLidFeederPackageState[2].bFormPresent	:= TRUE; //ok
		eBeforeLidFeederPackageState[1].bFormPresent	:= TRUE; //ok
		bWickFeederDragDelayAfterStartFullRegister		:= TRUE;
END_IF
	
(**Sorter**)
IF 	(eDispencersPackageState[1].bFormPresent AND eDispencersPackageState[1].bBottlePresent) OR	
	(eDispencersPackageState[2].bFormPresent AND eDispencersPackageState[2].bBottlePresent) OR	
	(eDispencersPackageState[3].bFormPresent AND eDispencersPackageState[3].bBottlePresent) OR		
	(eDispencersPackageState[4].bFormPresent AND eDispencersPackageState[4].bBottlePresent) OR		
	(eLidFeederPackageState[1].bFormPresent AND eLidFeederPackageState[1].bBottlePresent) 	OR		
	(eLidFeederPackageState[2].bFormPresent AND eLidFeederPackageState[2].bBottlePresent) 		
THEN
	VIS.bWickFeederSorterRun := TRUE;
END_IF

(**Prepare*)				
IF	bWickFeederDragingStationEnable AND 	tonLongDelayAfterStart.Q AND NOT P06_WickFeeder.fbWickFeederDragStation.bCycleDone AND
								fbIbLidFeederThirdFormCheckFormSensor.bOut AND 
								tonDelayAfterStart.Q AND 
								bWickFeederDragDelayAfterStartFullRegister AND iWickFeederDragCase = 10 AND
								NOT bWickFeederDragingStationPrepareRun AND NOT VIS.bWickFeederDragingStationRun AND
								P06_WickFeeder.fbWickFeederDragStation.eState = E_Station.eReady AND
								NOT tofbWickFeederDragingStationPrepareRun.Q

THEN
	bWickFeederDragingStationPrepareRun	:=	TRUE;
END_IF

IF (P00_PackML.fbPMLAuto.ePMLState = E_PMLState.ePMLState_STOPPING) THEN
	bWickFeederDragingStationPrepareRun	:=	FALSE;
END_IF

(*Drag*)
CASE iWickFeederDragCase OF
	0:
		IF bWickFeederDragingStationEnable AND tonLongDelayAfterStart.Q AND NOT VIS.bWickFeederDragingStationRun AND NOT P06_WickFeeder.fbWickFeederDragStation.bCycleDone AND VIS.bBarrierLidFeederRun AND
			P06_WickFeeder.fbWickFeederDragStation.eState = E_Station.eReady	
		THEN
			iWickFeederDragCase				:=	10;
		END_IF
	//Po staremu	
	10: 
		IF  (eBeforeLidFeederPackageState[1].bFormPresent AND eBeforeLidFeederPackageState[2].bFormPresent (*AND eBeforeLidFeeder2PackageState[1].bFormPresent*)) AND
			(eLidFeederPackageState[1].bLidPutted OR eLidFeederPackageState[1].bLidPutAborted OR NOT eLidFeederPackageState[1].bBottlePresent OR NOT eLidFeederPackageState[1].bLidPuttedOK) AND
			(eLidFeederPackageState[2].bLidPutted OR eLidFeederPackageState[2].bLidPutAborted OR NOT eLidFeederPackageState[2].bBottlePresent OR NOT eLidFeederPackageState[2].bLidPuttedOK) AND			
			tonLidFeederThirdFormsSensor.Q AND (bWickFeederReady OR NOT bWickFeederEnable) AND
			bWickFeederDragDelayAfterStartFullRegister AND 
			tonAfterWickFeederEmpty.Q AND
			NOT eAfterLidFeederPackageState[1].bFormPresent AND NOT eAfterLidFeederPackageState[2].bFormPresent AND
			(
			(NOT eBeforeLidSealerPackageState[1].bFormPresent AND NOT eBeforeLidSealerPackageState[2].bFormPresent) OR 
			(eBeforeLidSealerPackageState[1].bFormPresent AND eBeforeLidSealerPackageState[2].bFormPresent AND VIS.bLidSealerDragingStationRun)
			)
			AND
			fbIbLidFeederThirdFormCheckFormSensor.bOUT AND
			iWickFeederDragStoppingCount < 3 AND
			tonDelayAfterStart.Q AND 
			fbIbWickFeederAfterSensor.bOut AND
			tonbFormTransportersScrewerCmdStart.Q
		THEN 
			VIS.bWickFeederDragingStationRun	:=	TRUE;
			IF (P00_PackML.fbPMLAuto.ePMLState = E_PMLState.ePMLState_STOPPING)	THEN
				iWickFeederDragStoppingCount	:=	iWickFeederDragStoppingCount	+	1;
			END_IF
			iWickFeederDragCase				:=	20;
		END_IF
	20:
		iWickFeederDragCase:=25;

	25: 
		IF P06_WickFeeder.fbWickFeederDragStation.bCycleDone OR NOT VIS.bWickFeederDragingStationRun THEN
			iWickFeederDragCase:=30;
		END_IF
		
	30: // jak skonczylo zakręcanie to wroc do poczatku
		VIS.bWickFeederDragingStationRun					:=	FALSE;
		bWickFeederDragingStationPrepareRun			:=	FALSE;
		iWickFeederDragCase								:=	50;
	50:
		IF iWickFeederDragStoppingCount < 3 THEN
			iWickFeederDragCase:=0;	
		END_IF
END_CASE


(************************************)
//Deklaracja opóźnienia startu zakręcania
tonStartWickFeederDelay();
tonStartWickFeederDelay.IN:=	(P00_PackML.fbPMLAuto.ePMLState = E_PMLState.ePMLState_EXECUTE OR (P00_PackML.fbPMLAuto.ePMLState = E_PMLState.ePMLState_STOPPING AND iWickFeederDragStoppingCount < 3)) AND 
							((eLidFeederPackageState[1].bFormPresent) AND
							(NOT eLidFeederPackageState[1].bLidPutted AND NOT eLidFeederPackageState[1].bLidPutAborted )) AND
							((eLidFeederPackageState[2].bFormPresent) AND 
							(NOT eLidFeederPackageState[2].bLidPutted AND NOT eLidFeederPackageState[2].bLidPutAborted ))
;
tonStartWickFeederDelay.PT:=INT_TO_TIME(200);




IF bWickFeederEnable THEN
	

	CASE iWickFeederCase OF
		0:
			iWickFeederCase	:= 1;
	
		1: //Wykrywanie podjechania nowych wózków i opóźnienie
			IF	tonStartWickFeederDelay.Q AND tonDelayAfterStart.Q AND VIS.bBarrierLidFeederRun THEN	
				iWickFeederCase	:= 2;
			END_IF
			
		2:	//Rozpoczecie 
			IF (*tonDelayLid1Putting.q AND*) bWickFeederEnable AND eLidFeederPackageState[1].bBottlePresent AND eLidFeederPackageState[1].bWeightOK AND eLidFeederPackageState[1].nCardNumber > 0  
			THEN			
				VIS.bWickFeeder1Run 										:=	TRUE;
			END_IF
				
			IF (*tonDelayLid2Putting.q AND*) bWickFeederEnable AND eLidFeederPackageState[2].bBottlePresent AND eLidFeederPackageState[2].bWeightOK AND eLidFeederPackageState[2].nCardNumber > 0 
			THEN			
				VIS.bWickFeeder2Run 										:=	TRUE;
			END_IF
			iWickFeederCase	:= 3;
			
		3: //Czekanie na koniec 	
			//Warunek przejścia dalej, albo wykonano zakręcanie albo nie było rozkazu zakręcania (np. brak butelki)
			IF (
				VIS.bWickFeeder1Run AND (P06_WickFeeder.fbWickFeederSt.bCycleDone1 OR P06_WickFeeder.fbWickFeederSt.bCycleNotDone1)
				OR NOT VIS.bWickFeeder1Run
				) 
				AND
				(
				VIS.bWickFeeder2Run AND (P06_WickFeeder.fbWickFeederSt.bCycleDone2 OR P06_WickFeeder.fbWickFeederSt.bCycleNotDone2)
				OR NOT VIS.bWickFeeder2Run
				)
				THEN
					iWickFeederCase	:= 4;
			END_IF
		
		4: //Zapisywanie rejestrów i kasowanie sygnałów

			eLidFeederPackageState[1].tLidPuttingTime 				:=	P06_WickFeeder.fbWickFeederSt.tCycleTime;
			eLidFeederPackageState[2].tLidPuttingTime 				:=	P06_WickFeeder.fbWickFeederSt.tCycleTime;		
			
			IF P06_WickFeeder.fbWickFeederSt.bCycleDone1 THEN
				eLidFeederPackageState[1].bLidPutted 				:=	TRUE;
			ELSIF P06_WickFeeder.fbWickFeederSt.bCycleNotDone1 THEN
				eLidFeederPackageState[1].bLidPutted				:=	FALSE;
				eLidFeederPackageState[1].bLidPutAborted			:=	TRUE;
			ELSIF NOT bWickFeederEnable THEN
				eLidFeederPackageState[1].bLidPutted				:=	TRUE;
			ELSE // Jak wyłączona
				eLidFeederPackageState[1].bLidPutted				:=	TRUE; 
				eLidFeederPackageState[1].bLidPutAborted			:=	TRUE;
			END_IF

			IF P06_WickFeeder.fbWickFeederSt.bCycleDone2 THEN
				eLidFeederPackageState[2].bLidPutted 				:=	TRUE;
			ELSIF P06_WickFeeder.fbWickFeederSt.bCycleNotDone2 THEN
				eLidFeederPackageState[2].bLidPutted				:=	FALSE;
				eLidFeederPackageState[2].bLidPutAborted			:=	TRUE;
			ELSIF NOT bWickFeederEnable THEN
				eLidFeederPackageState[2].bLidPutted				:=	TRUE;
			ELSE // Jak wyłączona
				eLidFeederPackageState[2].bLidPutted				:=	TRUE; 
				eLidFeederPackageState[2].bLidPutAborted			:=	TRUE;
			END_IF
						
			FOR y:=1 TO 100 DO
				IF  eRFID[y].nCardNumber=eLidFeederPackageState[1].nCardNumber AND eLidFeederPackageState[1].nCardNumber >0 THEN
				 eRFID[y]:=eLidFeederPackageState[1];
				 EXIT;
				 END_IF;
			END_FOR
			 
			FOR z:=1 TO 100 DO
				IF  eRFID[z].nCardNumber=eLidFeederPackageState[2].nCardNumber AND eLidFeederPackageState[2].nCardNumber >0 THEN
					eRFID[z]:=eLidFeederPackageState[2];
				 EXIT;
				END_IF;
			END_FOR 
			 	
			 iWickFeederCase := 5; 
			 
		5: 
			VIS.bWickFeeder1PrepareRun 									:=	FALSE;	
			VIS.bWickFeeder2PrepareRun 									:=	FALSE;		
			VIS.bWickFeeder1Run 										:=	FALSE;	
			VIS.bWickFeeder2Run 										:=	FALSE;
			

			(***Nie wykonuj dalej ruchu gdy wcisnięty stop lub błąd***)
			IF NOT (P00_PackML.fbPMLAuto.ePMLState = E_PMLState.ePMLState_STOPPING) OR iWickFeederDragStoppingCount < 3 THEN
				iWickFeederCase := 0;
			END_IF
			
	END_CASE
ELSE
	eLidFeederPackageState[1].bLidPutted 				:=	TRUE;
	eLidFeederPackageState[2].bLidPutted 				:=	TRUE;	
	
	FOR y:=1 TO 100 DO
		IF  eRFID[y].nCardNumber=eLidFeederPackageState[1].nCardNumber AND eLidFeederPackageState[1].nCardNumber >0 THEN
			 eRFID[y]:=eLidFeederPackageState[1];
		EXIT;
		END_IF;
	 END_FOR
			 
